gfCNCPoint5[8465] = {X 489.4800, Y 58.0000, Z -7.1667, A 0.000, B 0.000, C 0.000 }
gfCNCPoint5[8466] = {X 489.4795, Y 59.0537, Z -7.1667, A 0.000, B 0.000, C 0.000 }
gfCNCPoint5[8467] = {X 489.3596, Y 60.7976, Z -7.1667, A 0.000, B 0.000, C 0.000 }
gfCNCPoint5[8468] = {X 489.0304, Y 62.5143, Z -7.1667, A 0.000, B 0.000, C 0.000 }
gfCNCPoint5[8469] = {X 488.4968, Y 64.1788, Z -7.1667, A 0.000, B 0.000, C 0.000 }
gfCNCPoint5[8470] = {X 487.7665, Y 65.7669, Z -7.1667, A 0.000, B 0.000, C 0.000 }
gfCNCPoint5[8471] = {X 486.8501, Y 67.2554, Z -7.1667, A 0.000, B 0.000, C 0.000 }
gfCNCPoint5[8472] = {X 485.7611, Y 68.6227, Z -7.1667, A 0.000, B 0.000, C 0.000 }
gfCNCPoint5[8473] = {X 485.7614, Y 87.3811, Z -7.1667, A 0.000, B 0.000, C 0.000 }
gfCNCPoint5[8474] = {X 486.0686, Y 87.7333, Z -7.1667, A 0.000, B 0.000, C 0.000 }
gfCNCPoint5[8475] = {X 486.3643, Y 88.0951, Z -7.1667, A 0.000, B 0.000, C 0.000 }
gfCNCPoint5[8476] = {X 507.6812, Y 88.0951, Z -7.1667, A 0.000, B 0.000, C 0.000 }
gfCNCPoint5[8477] = {X 507.6812, Y 90.4951, Z -7.1667, A 0.000, B 0.000, C 0.000 }
gfCNCPoint5[8478] = {X 590.4967, Y 90.4951, Z -7.1667, A 0.000, B 0.000, C 0.000 }
gfCNCPoint5[8479] = {X 590.4967, Y 58.6615, Z -7.1667, A 0.000, B 0.000, C 0.000 }
gfCNCPoint5[8480] = {X 588.9715, Y 58.2279, Z -7.1667, A 0.000, B 0.000, C 0.000 }
gfCNCPoint5[8481] = {X 587.5052, Y 57.6246, Z -7.1667, A 0.000, B 0.000, C 0.000 }
gfCNCPoint5[8482] = {X 585.8387, Y 58.2956, Z -7.1667, A 0.000, B 0.000, C 0.000 }
gfCNCPoint5[8483] = {X 584.0999, Y 58.7477, Z -7.1667, A 0.000, B 0.000, C 0.000 }
gfCNCPoint5[8484] = {X 582.3176, Y 58.9733, Z -7.1667, A 0.000, B 0.000, C 0.000 }
gfCNCPoint5[8485] = {X 580.5210, Y 58.9689, Z -7.1667, A 0.000, B 0.000, C 0.000 }
gfCNCPoint5[8486] = {X 578.7398, Y 58.7344, Z -7.1667, A 0.000, B 0.000, C 0.000 }
gfCNCPoint5[8487] = {X 577.0034, Y 58.2738, Z -7.1667, A 0.000, B 0.000, C 0.000 }
gfCNCPoint5[8488] = {X 575.3401, Y 57.5945, Z -7.1667, A 0.000, B 0.000, C 0.000 }
gfCNCPoint5[8489] = {X 573.8813, Y 58.2035, Z -7.1667, A 0.000, B 0.000, C 0.000 }
gfCNCPoint5[8490] = {X 572.3630, Y 58.6441, Z -7.1667, A 0.000, B 0.000, C 0.000 }
gfCNCPoint5[8491] = {X 570.8048, Y 58.9107, Z -7.1667, A 0.000, B 0.000, C 0.000 }
gfCNCPoint5[8492] = {X 569.2264, Y 59.0000, Z -7.1667, A 0.000, B 0.000, C 0.000 }
gfCNCPoint5[8493] = {X 562.4443, Y 59.0000, Z -7.1667, A 0.000, B 0.000, C 0.000 }
gfCNCPoint5[8494] = {X 560.6169, Y 58.8802, Z -7.1667, A 0.000, B 0.000, C 0.000 }
gfCNCPoint5[8495] = {X 558.8208, Y 58.5230, Z -7.1667, A 0.000, B 0.000, C 0.000 }
gfCNCPoint5[8496] = {X 557.0867, Y 57.9343, Z -7.1667, A 0.000, B 0.000, C 0.000 }
gfCNCPoint5[8497] = {X 555.4443, Y 57.1244, Z -7.1667, A 0.000, B 0.000, C 0.000 }
gfCNCPoint5[8498] = {X 553.9216, Y 56.1069, Z -7.1667, A 0.000, B 0.000, C 0.000 }
gfCNCPoint5[8499] = {X 552.5448, Y 54.8995, Z -7.1667, A 0.000, B 0.000, C 0.000 }
gfCNCPoint5[8500] = {X 551.4383, Y 53.6527, Z -7.1667, A 0.000, B 0.000, C 0.000 }
gfCNCPoint5[8501] = {X 550.4879, Y 52.2832, Z -7.1667, A 0.000, B 0.000, C 0.000 }
gfCNCPoint5[8502] = {X 549.8381, Y 51.0896, Z -7.1667, A 0.000, B 0.000, C 0.000 }
gfCNCPoint5[8503] = {X 549.3070, Y 49.8386, Z -7.1667, A 0.000, B 0.000, C 0.000 }
gfCNCPoint5[8504] = {X 548.3757, Y 50.7155, Z -7.1667, A 0.000, B 0.000, C 0.000 }
gfCNCPoint5[8505] = {X 547.3054, Y 51.4159, Z -7.1667, A 0.000, B 0.000, C 0.000 }
gfCNCPoint5[8506] = {X 546.1638, Y 51.9069, Z -7.1667, A 0.000, B 0.000, C 0.000 }
gfCNCPoint5[8507] = {X 544.9553, Y 52.1968, Z -7.1667, A 0.000, B 0.000, C 0.000 }
gfCNCPoint5[8508] = {X 543.7151, Y 52.2769, Z -7.1667, A 0.000, B 0.000, C 0.000 }
gfCNCPoint5[8509] = {X 525.3425, Y 52.2772, Z -7.1667, A 0.000, B 0.000, C 0.000 }
gfCNCPoint5[8510] = {X 524.2751, Y 53.0687, Z -7.1667, A 0.000, B 0.000, C 0.000 }
gfCNCPoint5[8511] = {X 523.0839, Y 53.6575, Z -7.1667, A 0.000, B 0.000, C 0.000 }
gfCNCPoint5[8512] = {X 521.8069, Y 54.0249, Z -7.1667, A 0.000, B 0.000, C 0.000 }
gfCNCPoint5[8513] = {X 520.4849, Y 54.1591, Z -7.1667, A 0.000, B 0.000, C 0.000 }
gfCNCPoint5[8514] = {X 519.7998, Y 54.1591, Z -7.1667, A 0.000, B 0.000, C 0.000 }
gfCNCPoint5[8515] = {X 518.5529, Y 54.0515, Z -7.1667, A 0.000, B 0.000, C 0.000 }
gfCNCPoint5[8516] = {X 517.3428, Y 53.7320, Z -7.1667, A 0.000, B 0.000, C 0.000 }
gfCNCPoint5[8517] = {X 516.2054, Y 53.2099, Z -7.1667, A 0.000, B 0.000, C 0.000 }
gfCNCPoint5[8518] = {X 515.1742, Y 52.5007, Z -7.1667, A 0.000, B 0.000, C 0.000 }
gfCNCPoint5[8519] = {X 514.2797, Y 51.6254, Z -7.1667, A 0.000, B 0.000, C 0.000 }
gfCNCPoint5[8520] = {X 513.5483, Y 50.6098, Z -7.1667, A 0.000, B 0.000, C 0.000 }
gfCNCPoint5[8521] = {X 513.0017, Y 49.4839, Z -7.1667, A 0.000, B 0.000, C 0.000 }
gfCNCPoint5[8522] = {X 512.7353, Y 48.6374, Z -7.1667, A 0.000, B 0.000, C 0.000 }
gfCNCPoint5[8523] = {X 512.5739, Y 47.7649, Z -7.1667, A 0.000, B 0.000, C 0.000 }
gfCNCPoint5[8524] = {X 512.5198, Y 46.8791, Z -7.1667, A 0.000, B 0.000, C 0.000 }
gfCNCPoint5[8525] = {X 512.5198, Y 39.9011, Z -7.1667, A 0.000, B 0.000, C 0.000 }
gfCNCPoint5[8526] = {X 512.5808, Y 38.9604, Z -7.1667, A 0.000, B 0.000, C 0.000 }
gfCNCPoint5[8527] = {X 512.7629, Y 38.0355, Z -7.1667, A 0.000, B 0.000, C 0.000 }
gfCNCPoint5[8528] = {X 513.0629, Y 37.1419, Z -7.1667, A 0.000, B 0.000, C 0.000 }
gfCNCPoint5[8529] = {X 513.5586, Y 36.1533, Z -7.1667, A 0.000, B 0.000, C 0.000 }
gfCNCPoint5[8530] = {X 514.1983, Y 35.2512, Z -7.1667, A 0.000, B 0.000, C 0.000 }
gfCNCPoint5[8531] = {X 514.9672, Y 34.4564, Z -7.1667, A 0.000, B 0.000, C 0.000 }
gfCNCPoint5[8532] = {X 515.8477, Y 33.7872, Z -7.1667, A 0.000, B 0.000, C 0.000 }
gfCNCPoint5[8533] = {X 513.2419, Y 29.7561, Z -7.1667, A 0.000, B 0.000, C 0.000 }
gfCNCPoint5[8534] = {X 513.5220, Y 29.5804, Z -7.1667, A 0.000, B 0.000, C 0.000 }
gfCNCPoint5[8535] = {X 513.8068, Y 29.4125, Z -7.1667, A 0.000, B 0.000, C 0.000 }
gfCNCPoint5[8536] = {X 513.8068, Y 27.6757, Z -7.1667, A 0.000, B 0.000, C 0.000 }
gfCNCPoint5[8537] = {X 513.5219, Y 27.5014, Z -7.1667, A 0.000, B 0.000, C 0.000 }
gfCNCPoint5[8538] = {X 513.2419, Y 27.3192, Z -7.1667, A 0.000, B 0.000, C 0.000 }
gfCNCPoint5[8539] = {X 513.2419, Y 29.7561, Z -7.1667, A 0.000, B 0.000, C 0.000 }
gfCNCPoint5[8540] = {X 514.5448, Y 31.7717, Z -7.1667, A 0.000, B 0.000, C 0.000 }
gfCNCPoint5[8541] = {X 515.3550, Y 31.3019, Z -7.1667, A 0.000, B 0.000, C 0.000 }
gfCNCPoint5[8542] = {X 516.2068, Y 30.9126, Z -7.1667, A 0.000, B 0.000, C 0.000 }
gfCNCPoint5[8543] = {X 516.2068, Y 26.2046, Z -7.1667, A 0.000, B 0.000, C 0.000 }
gfCNCPoint5[8544] = {X 515.3716, Y 25.8042, Z -7.1667, A 0.000, B 0.000, C 0.000 }
gfCNCPoint5[8545] = {X 514.5784, Y 25.3258, Z -7.1667, A 0.000, B 0.000, C 0.000 }
gfCNCPoint5[8546] = {X 513.5954, Y 24.5712, Z -7.1667, A 0.000, B 0.000, C 0.000 }
gfCNCPoint5[8547] = {X 512.7167, Y 23.6971, Z -7.1667, A 0.000, B 0.000, C 0.000 }
gfCNCPoint5[8548] = {X 511.9570, Y 22.7179, Z -7.1667, A 0.000, B 0.000, C 0.000 }
gfCNCPoint5[8549] = {X 511.3286, Y 21.6497, Z -7.1667, A 0.000, B 0.000, C 0.000 }
gfCNCPoint5[8550] = {X 510.8418, Y 20.5099, Z -7.1667, A 0.000, B 0.000, C 0.000 }
gfCNCPoint5[8551] = {X 510.8420, Y 36.2322, Z -7.1667, A 0.000, B 0.000, C 0.000 }
gfCNCPoint5[8552] = {X 511.5011, Y 34.9177, Z -7.1667, A 0.000, B 0.000, C 0.000 }
gfCNCPoint5[8553] = {X 512.3517, Y 33.7182, Z -7.1667, A 0.000, B 0.000, C 0.000 }
gfCNCPoint5[8554] = {X 513.3741, Y 32.6614, Z -7.1667, A 0.000, B 0.000, C 0.000 }
gfCNCPoint5[8555] = {X 514.5448, Y 31.7717, Z -7.1667, A 0.000, B 0.000, C 0.000 }
gfCNCPoint5[8556] = {X 515.8477, Y 33.7872, Z -7.1667, A 0.000, B 0.000, C 0.000 }
gfCNCPoint5[8557] = {X 516.7441, Y 33.2935, Z -7.1667, A 0.000, B 0.000, C 0.000 }
gfCNCPoint5[8558] = {X 517.7008, Y 32.9303, Z -7.1667, A 0.000, B 0.000, C 0.000 }
gfCNCPoint5[8559] = {X 518.6990, Y 32.7048, Z -7.1667, A 0.000, B 0.000, C 0.000 }
gfCNCPoint5[8560] = {X 518.6299, Y 32.1290, Z -7.1667, A 0.000, B 0.000, C 0.000 }
gfCNCPoint5[8561] = {X 518.6068, Y 31.5494, Z -7.1667, A 0.000, B 0.000, C 0.000 }
gfCNCPoint5[8562] = {X 518.6068, Y 24.5714, Z -7.1667, A 0.000, B 0.000, C 0.000 }
gfCNCPoint5[8563] = {X 518.6080, Y 24.4373, Z -7.1667, A 0.000, B 0.000, C 0.000 }
gfCNCPoint5[8564] = {X 517.3914, Y 24.0941, Z -7.1667, A 0.000, B 0.000, C 0.000 }
gfCNCPoint5[8565] = {X 516.2525, Y 23.5455, Z -7.1667, A 0.000, B 0.000, C 0.000 }
gfCNCPoint5[8566] = {X 515.2257, Y 22.8082, Z -7.1667, A 0.000, B 0.000, C 0.000 }
gfCNCPoint5[8567] = {X 514.3419, Y 21.9045, Z -7.1667, A 0.000, B 0.000, C 0.000 }
gfCNCPoint5[8568] = {X 513.6277, Y 20.8614, Z -7.1667, A 0.000, B 0.000, C 0.000 }
gfCNCPoint5[8569] = {X 513.1048, Y 19.7105, Z -7.1667, A 0.000, B 0.000, C 0.000 }
gfCNCPoint5[8570] = {X 512.7938, Y 18.5158, Z -7.1667, A 0.000, B 0.000, C 0.000 }
gfCNCPoint5[8571] = {X 512.6891, Y 17.2857, Z -7.1667, A 0.000, B 0.000, C 0.000 }
gfCNCPoint5[8572] = {X 512.6891, Y 10.3077, Z -7.1667, A 0.000, B 0.000, C 0.000 }
gfCNCPoint5[8573] = {X 512.7002, Y 9.9057, Z -7.1667, A 0.000, B 0.000, C 0.000 }
gfCNCPoint5[8574] = {X 512.7335, Y 9.5049, Z -7.1667, A 0.000, B 0.000, C 0.000 }
gfCNCPoint5[8575] = {X 509.4593, Y 9.5049, Z -7.1667, A 0.000, B 0.000, C 0.000 }
gfCNCPoint5[8576] = {X 509.7407, Y 10.3716, Z -7.1667, A 0.000, B 0.000, C 0.000 }
gfCNCPoint5[8577] = {X 509.9113, Y 11.2668, Z -7.1667, A 0.000, B 0.000, C 0.000 }
gfCNCPoint5[8578] = {X 509.9685, Y 12.1762, Z -7.1667, A 0.000, B 0.000, C 0.000 }
gfCNCPoint5[8579] = {X 509.9682, Y 13.0462, Z -7.1667, A 0.000, B 0.000, C 0.000 }
gfCNCPoint5[8580] = {X 509.8612, Y 14.2233, Z -7.1667, A 0.000, B 0.000, C 0.000 }
gfCNCPoint5[8581] = {X 509.5651, Y 15.3676, Z -7.1667, A 0.000, B 0.000, C 0.000 }
gfCNCPoint5[8582] = {X 509.0878, Y 16.4489, Z -7.1667, A 0.000, B 0.000, C 0.000 }
gfCNCPoint5[8583] = {X 508.4418, Y 17.4387, Z -7.1667, A 0.000, B 0.000, C 0.000 }
gfCNCPoint5[8584] = {X 508.4420, Y 39.7484, Z -7.1667, A 0.000, B 0.000, C 0.000 }
gfCNCPoint5[8585] = {X 509.0898, Y 40.7415, Z -7.1667, A 0.000, B 0.000, C 0.000 }
gfCNCPoint5[8586] = {X 509.5677, Y 41.8266, Z -7.1667, A 0.000, B 0.000, C 0.000 }
gfCNCPoint5[8587] = {X 509.8632, Y 42.9748, Z -7.1667, A 0.000, B 0.000, C 0.000 }
gfCNCPoint5[8588] = {X 509.9683, Y 44.1558, Z -7.1667, A 0.000, B 0.000, C 0.000 }
gfCNCPoint5[8589] = {X 509.9685, Y 45.0000, Z -7.1667, A 0.000, B 0.000, C 0.000 }
gfCNCPoint5[8590] = {X 509.8909, Y 46.0603, Z -7.1667, A 0.000, B 0.000, C 0.000 }
gfCNCPoint5[8591] = {X 509.6596, Y 47.0980, Z -7.1667, A 0.000, B 0.000, C 0.000 }
gfCNCPoint5[8592] = {X 509.2797, Y 48.0910, Z -7.1667, A 0.000, B 0.000, C 0.000 }
gfCNCPoint5[8593] = {X 508.7593, Y 49.0180, Z -7.1667, A 0.000, B 0.000, C 0.000 }
gfCNCPoint5[8594] = {X 508.0200, Y 49.9571, Z -7.1667, A 0.000, B 0.000, C 0.000 }
gfCNCPoint5[8595] = {X 507.1371, Y 50.7626, Z -7.1667, A 0.000, B 0.000, C 0.000 }
gfCNCPoint5[8596] = {X 506.1343, Y 51.4129, Z -7.1667, A 0.000, B 0.000, C 0.000 }
gfCNCPoint5[8597] = {X 505.0386, Y 51.8902, Z -7.1667, A 0.000, B 0.000, C 0.000 }
gfCNCPoint5[8598] = {X 503.8796, Y 52.1819, Z -7.1667, A 0.000, B 0.000, C 0.000 }
gfCNCPoint5[8599] = {X 502.6885, Y 52.2800, Z -7.1667, A 0.000, B 0.000, C 0.000 }
gfCNCPoint5[8600] = {X 496.2450, Y 52.2800, Z -7.1667, A 0.000, B 0.000, C 0.000 }
gfCNCPoint5[8601] = {X 495.0845, Y 52.1869, Z -7.1667, A 0.000, B 0.000, C 0.000 }
gfCNCPoint5[8602] = {X 493.9538, Y 51.9100, Z -7.1667, A 0.000, B 0.000, C 0.000 }
gfCNCPoint5[8603] = {X 492.8816, Y 51.4564, Z -7.1667, A 0.000, B 0.000, C 0.000 }
gfCNCPoint5[8604] = {X 491.8954, Y 50.8377, Z -7.1667, A 0.000, B 0.000, C 0.000 }
gfCNCPoint5[8605] = {X 491.0204, Y 50.0697, Z -7.1667, A 0.000, B 0.000, C 0.000 }
gfCNCPoint5[8606] = {X 490.2980, Y 49.1989, Z -7.1667, A 0.000, B 0.000, C 0.000 }
gfCNCPoint5[8607] = {X 489.7192, Y 48.2267, Z -7.1667, A 0.000, B 0.000, C 0.000 }
gfCNCPoint5[8608] = {X 489.2980, Y 47.1766, Z -7.1667, A 0.000, B 0.000, C 0.000 }
gfCNCPoint5[8609] = {X 488.8769, Y 48.2267, Z -7.1667, A 0.000, B 0.000, C 0.000 }
gfCNCPoint5[8610] = {X 488.2981, Y 49.1989, Z -7.1667, A 0.000, B 0.000, C 0.000 }
gfCNCPoint5[8611] = {X 487.5756, Y 50.0697, Z -7.1667, A 0.000, B 0.000, C 0.000 }
gfCNCPoint5[8612] = {X 486.8824, Y 50.6978, Z -7.1667, A 0.000, B 0.000, C 0.000 }
gfCNCPoint5[8613] = {X 486.1145, Y 51.2318, Z -7.1667, A 0.000, B 0.000, C 0.000 }
gfCNCPoint5[8614] = {X 485.2843, Y 51.6629, Z -7.1667, A 0.000, B 0.000, C 0.000 }
gfCNCPoint5[8615] = {X 486.0586, Y 53.1385, Z -7.1667, A 0.000, B 0.000, C 0.000 }
gfCNCPoint5[8616] = {X 486.6224, Y 54.7067, Z -7.1667, A 0.000, B 0.000, C 0.000 }
gfCNCPoint5[8617] = {X 486.9651, Y 56.3375, Z -7.1667, A 0.000, B 0.000, C 0.000 }
gfCNCPoint5[8618] = {X 487.0800, Y 58.0000, Z -7.1667, A 0.000, B 0.000, C 0.000 }
gfCNCPoint5[8619] = {X 487.0796, Y 59.0339, Z -7.1667, A 0.000, B 0.000, C 0.000 }
gfCNCPoint5[8620] = {X 486.9596, Y 60.6350, Z -7.1667, A 0.000, B 0.000, C 0.000 }
gfCNCPoint5[8621] = {X 486.6284, Y 62.2061, Z -7.1667, A 0.000, B 0.000, C 0.000 }
gfCNCPoint5[8622] = {X 486.0918, Y 63.7194, Z -7.1667, A 0.000, B 0.000, C 0.000 }
gfCNCPoint5[8623] = {X 485.3591, Y 65.1481, Z -7.1667, A 0.000, B 0.000, C 0.000 }
gfCNCPoint5[8624] = {X 484.4435, Y 66.4671, Z -7.1667, A 0.000, B 0.000, C 0.000 }
gfCNCPoint5[8625] = {X 483.3611, Y 67.6530, Z -7.1667, A 0.000, B 0.000, C 0.000 }
gfCNCPoint5[8626] = {X 483.3614, Y 88.3518, Z -7.1667, A 0.000, B 0.000, C 0.000 }
gfCNCPoint5[8627] = {X 484.3105, Y 89.3721, Z -7.1667, A 0.000, B 0.000, C 0.000 }
gfCNCPoint5[8628] = {X 485.1356, Y 90.4951, Z -7.1667, A 0.000, B 0.000, C 0.000 }
gfCNCPoint5[8629] = {X 507.6812, Y 90.4951, Z -7.1667, A 0.000, B 0.000, C 0.000 }
gfCNCPoint5[8630] = {X 507.6812, Y 92.8951, Z -7.1667, A 0.000, B 0.000, C 0.000 }
gfCNCPoint5[8631] = {X 592.8967, Y 92.8951, Z -7.1667, A 0.000, B 0.000, C 0.000 }
gfCNCPoint5[8632] = {X 592.8967, Y 56.5812, Z -7.1667, A 0.000, B 0.000, C 0.000 }
gfCNCPoint5[8633] = {X 591.4811, Y 56.4128, Z -7.1667, A 0.000, B 0.000, C 0.000 }
gfCNCPoint5[8634] = {X 590.0968, Y 56.0721, Z -7.1667, A 0.000, B 0.000, C 0.000 }
gfCNCPoint5[8635] = {X 588.7648, Y 55.5641, Z -7.1667, A 0.000, B 0.000, C 0.000 }
gfCNCPoint5[8636] = {X 587.5052, Y 54.8965, Z -7.1667, A 0.000, B 0.000, C 0.000 }
gfCNCPoint5[8637] = {X 586.9690, Y 55.2051, Z -7.1667, A 0.000, B 0.000, C 0.000 }
gfCNCPoint5[8638] = {X 586.4171, Y 55.4846, Z -7.1667, A 0.000, B 0.000, C 0.000 }
gfCNCPoint5[8639] = {X 584.8782, Y 56.0830, Z -7.1667, A 0.000, B 0.000, C 0.000 }
gfCNCPoint5[8640] = {X 583.2699, Y 56.4570, Z -7.1667, A 0.000, B 0.000, C 0.000 }
gfCNCPoint5[8641] = {X 581.6248, Y 56.5987, Z -7.1667, A 0.000, B 0.000, C 0.000 }
gfCNCPoint5[8642] = {X 579.9763, Y 56.5055, Z -7.1667, A 0.000, B 0.000, C 0.000 }
gfCNCPoint5[8643] = {X 578.3577, Y 56.1792, Z -7.1667, A 0.000, B 0.000, C 0.000 }
gfCNCPoint5[8644] = {X 576.8018, Y 55.6263, Z -7.1667, A 0.000, B 0.000, C 0.000 }
gfCNCPoint5[8645] = {X 575.3401, Y 54.8581, Z -7.1667, A 0.000, B 0.000, C 0.000 }
gfCNCPoint5[8646] = {X 573.9176, Y 55.6091, Z -7.1667, A 0.000, B 0.000, C 0.000 }
gfCNCPoint5[8647] = {X 572.4049, Y 56.1560, Z -7.1667, A 0.000, B 0.000, C 0.000 }
gfCNCPoint5[8648] = {X 570.8311, Y 56.4885, Z -7.1667, A 0.000, B 0.000, C 0.000 }
gfCNCPoint5[8649] = {X 569.2264, Y 56.6000, Z -7.1667, A 0.000, B 0.000, C 0.000 }
gfCNCPoint5[8650] = {X 562.4443, Y 56.6000, Z -7.1667, A 0.000, B 0.000, C 0.000 }
gfCNCPoint5[8651] = {X 560.9302, Y 56.5008, Z -7.1667, A 0.000, B 0.000, C 0.000 }
gfCNCPoint5[8652] = {X 559.4420, Y 56.2047, Z -7.1667, A 0.000, B 0.000, C 0.000 }
gfCNCPoint5[8653] = {X 558.0052, Y 55.7170, Z -7.1667, A 0.000, B 0.000, C 0.000 }
gfCNCPoint5[8654] = {X 556.6443, Y 55.0459, Z -7.1667, A 0.000, B 0.000, C 0.000 }
gfCNCPoint5[8655] = {X 555.3827, Y 54.2029, Z -7.1667, A 0.000, B 0.000, C 0.000 }
gfCNCPoint5[8656] = {X 554.2419, Y 53.2024, Z -7.1667, A 0.000, B 0.000, C 0.000 }
gfCNCPoint5[8657] = {X 553.4046, Y 52.2694, Z -7.1667, A 0.000, B 0.000, C 0.000 }
gfCNCPoint5[8658] = {X 552.6729, Y 51.2514, Z -7.1667, A 0.000, B 0.000, C 0.000 }
gfCNCPoint5[8659] = {X 552.0553, Y 50.1604, Z -7.1667, A 0.000, B 0.000, C 0.000 }
gfCNCPoint5[8660] = {X 551.5591, Y 49.0091, Z -7.1667, A 0.000, B 0.000, C 0.000 }
gfCNCPoint5[8661] = {X 551.1638, Y 47.7039, Z -7.1667, A 0.000, B 0.000, C 0.000 }
gfCNCPoint5[8662] = {X 550.9245, Y 46.3614, Z -7.1667, A 0.000, B 0.000, C 0.000 }
gfCNCPoint5[8663] = {X 550.8443, Y 45.0000, Z -7.1667, A 0.000, B 0.000, C 0.000 }
gfCNCPoint5[8664] = {X 550.8443, Y 44.0403, Z -7.1667, A 0.000, B 0.000, C 0.000 }
gfCNCPoint5[8665] = {X 550.9580, Y 42.4569, Z -7.1667, A 0.000, B 0.000, C 0.000 }
gfCNCPoint5[8666] = {X 551.2863, Y 40.9037, Z -7.1667, A 0.000, B 0.000, C 0.000 }
gfCNCPoint5[8667] = {X 551.8231, Y 39.4097, Z -7.1667, A 0.000, B 0.000, C 0.000 }
gfCNCPoint5[8668] = {X 549.6250, Y 38.4460, Z -7.1667, A 0.000, B 0.000, C 0.000 }
gfCNCPoint5[8669] = {X 549.7927, Y 38.0781, Z -7.1667, A 0.000, B 0.000, C 0.000 }
gfCNCPoint5[8670] = {X 549.9709, Y 37.7152, Z -7.1667, A 0.000, B 0.000, C 0.000 }
gfCNCPoint5[8671] = {X 549.9710, Y 16.9522, Z -7.1667, A 0.000, B 0.000, C 0.000 }
gfCNCPoint5[8672] = {X 549.8033, Y 17.1983, Z -7.1667, A 0.000, B 0.000, C 0.000 }
gfCNCPoint5[8673] = {X 549.6257, Y 17.4374, Z -7.1667, A 0.000, B 0.000, C 0.000 }
gfCNCPoint5[8674] = {X 549.6250, Y 38.4460, Z -7.1667, A 0.000, B 0.000, C 0.000 }
gfCNCPoint5[8675] = {X 551.8231, Y 39.4097, Z -7.1667, A 0.000, B 0.000, C 0.000 }
gfCNCPoint5[8676] = {X 552.0827, Y 38.8574, Z -7.1667, A 0.000, B 0.000, C 0.000 }
gfCNCPoint5[8677] = {X 552.3709, Y 38.3195, Z -7.1667, A 0.000, B 0.000, C 0.000 }
gfCNCPoint5[8678] = {X 552.3710, Y 11.6864, Z -7.1667, A 0.000, B 0.000, C 0.000 }
gfCNCPoint5[8679] = {X 551.6701, Y 10.2325, Z -7.1667, A 0.000, B 0.000, C 0.000 }
gfCNCPoint5[8680] = {X 551.1778, Y 8.6954, Z -7.1667, A 0.000, B 0.000, C 0.000 }
gfCNCPoint5[8681] = {X 550.9035, Y 7.1049, Z -7.1667, A 0.000, B 0.000, C 0.000 }
gfCNCPoint5[8682] = {X 524.2927, Y 7.1049, Z -7.1667, A 0.000, B 0.000, C 0.000 }
gfCNCPoint5[8683] = {X 524.3782, Y 7.2059, Z -7.1667, A 0.000, B 0.000, C 0.000 }
gfCNCPoint5[8684] = {X 524.4609, Y 7.3092, Z -7.1667, A 0.000, B 0.000, C 0.000 }
gfCNCPoint5[8685] = {X 543.7426, Y 7.3096, Z -7.1667, A 0.000, B 0.000, C 0.000 }
gfCNCPoint5[8686] = {X 544.7121, Y 7.3817, Z -7.1667, A 0.000, B 0.000, C 0.000 }
gfCNCPoint5[8687] = {X 545.6480, Y 7.6444, Z -7.1667, A 0.000, B 0.000, C 0.000 }
gfCNCPoint5[8688] = {X 546.5134, Y 8.0872, Z -7.1667, A 0.000, B 0.000, C 0.000 }
gfCNCPoint5[8689] = {X 547.2740, Y 8.6926, Z -7.1667, A 0.000, B 0.000, C 0.000 }
gfCNCPoint5[8690] = {X 547.8996, Y 9.4366, Z -7.1667, A 0.000, B 0.000, C 0.000 }
gfCNCPoint5[8691] = {X 548.3656, Y 10.2898, Z -7.1667, A 0.000, B 0.000, C 0.000 }
gfCNCPoint5[8692] = {X 548.6533, Y 11.2184, Z -7.1667, A 0.000, B 0.000, C 0.000 }
gfCNCPoint5[8693] = {X 548.7514, Y 12.1856, Z -7.1667, A 0.000, B 0.000, C 0.000 }
gfCNCPoint5[8694] = {X 548.7512, Y 13.0237, Z -7.1667, A 0.000, B 0.000, C 0.000 }
gfCNCPoint5[8695] = {X 548.6554, Y 13.9414, Z -7.1667, A 0.000, B 0.000, C 0.000 }
gfCNCPoint5[8696] = {X 548.3885, Y 14.8247, Z -7.1667, A 0.000, B 0.000, C 0.000 }
gfCNCPoint5[8697] = {X 547.9601, Y 15.6420, Z -7.1667, A 0.000, B 0.000, C 0.000 }
gfCNCPoint5[8698] = {X 547.6189, Y 16.1039, Z -7.1667, A 0.000, B 0.000, C 0.000 }
gfCNCPoint5[8699] = {X 547.2258, Y 16.5224, Z -7.1667, A 0.000, B 0.000, C 0.000 }
gfCNCPoint5[8700] = {X 547.2250, Y 40.6636, Z -7.1667, A 0.000, B 0.000, C 0.000 }
gfCNCPoint5[8701] = {X 547.8659, Y 41.4055, Z -7.1667, A 0.000, B 0.000, C 0.000 }
gfCNCPoint5[8702] = {X 548.3456, Y 42.2605, Z -7.1667, A 0.000, B 0.000, C 0.000 }
gfCNCPoint5[8703] = {X 548.6448, Y 43.1941, Z -7.1667, A 0.000, B 0.000, C 0.000 }
gfCNCPoint5[8704] = {X 548.7513, Y 44.1687, Z -7.1667, A 0.000, B 0.000, C 0.000 }
gfCNCPoint5[8705] = {X 548.7514, Y 45.0006, Z -7.1667, A 0.000, B 0.000, C 0.000 }
gfCNCPoint5[8706] = {X 548.6700, Y 45.8824, Z -7.1667, A 0.000, B 0.000, C 0.000 }
gfCNCPoint5[8707] = {X 548.4306, Y 46.7350, Z -7.1667, A 0.000, B 0.000, C 0.000 }
gfCNCPoint5[8708] = {X 548.0413, Y 47.5304, Z -7.1667, A 0.000, B 0.000, C 0.000 }
gfCNCPoint5[8709] = {X 547.5147, Y 48.2424, Z -7.1667, A 0.000, B 0.000, C 0.000 }
gfCNCPoint5[8710] = {X 546.7291, Y 48.9521, Z -7.1667, A 0.000, B 0.000, C 0.000 }
gfCNCPoint5[8711] = {X 545.8090, Y 49.4759, Z -7.1667, A 0.000, B 0.000, C 0.000 }
gfCNCPoint5[8712] = {X 544.7976, Y 49.7890, Z -7.1667, A 0.000, B 0.000, C 0.000 }
gfCNCPoint5[8713] = {X 543.7426, Y 49.8769, Z -7.1667, A 0.000, B 0.000, C 0.000 }
gfCNCPoint5[8714] = {X 524.3239, Y 49.8773, Z -7.1667, A 0.000, B 0.000, C 0.000 }
gfCNCPoint5[8715] = {X 523.7110, Y 50.5161, Z -7.1667, A 0.000, B 0.000, C 0.000 }
gfCNCPoint5[8716] = {X 522.9957, Y 51.0377, Z -7.1667, A 0.000, B 0.000, C 0.000 }
gfCNCPoint5[8717] = {X 522.2001, Y 51.4260, Z -7.1667, A 0.000, B 0.000, C 0.000 }
gfCNCPoint5[8718] = {X 521.3488, Y 51.6690, Z -7.1667, A 0.000, B 0.000, C 0.000 }
gfCNCPoint5[8719] = {X 520.4681, Y 51.7591, Z -7.1667, A 0.000, B 0.000, C 0.000 }
gfCNCPoint5[8720] = {X 519.7998, Y 51.7591, Z -7.1667, A 0.000, B 0.000, C 0.000 }
gfCNCPoint5[8721] = {X 518.8477, Y 51.6654, Z -7.1667, A 0.000, B 0.000, C 0.000 }
gfCNCPoint5[8722] = {X 517.9323, Y 51.3877, Z -7.1667, A 0.000, B 0.000, C 0.000 }
gfCNCPoint5[8723] = {X 517.0886, Y 50.9367, Z -7.1667, A 0.000, B 0.000, C 0.000 }
gfCNCPoint5[8724] = {X 516.3491, Y 50.3298, Z -7.1667, A 0.000, B 0.000, C 0.000 }
gfCNCPoint5[8725] = {X 515.7422, Y 49.5903, Z -7.1667, A 0.000, B 0.000, C 0.000 }
gfCNCPoint5[8726] = {X 515.2912, Y 48.7466, Z -7.1667, A 0.000, B 0.000, C 0.000 }
gfCNCPoint5[8727] = {X 515.0135, Y 47.8312, Z -7.1667, A 0.000, B 0.000, C 0.000 }
gfCNCPoint5[8728] = {X 514.9198, Y 46.8791, Z -7.1667, A 0.000, B 0.000, C 0.000 }
gfCNCPoint5[8729] = {X 514.9198, Y 39.9011, Z -7.1667, A 0.000, B 0.000, C 0.000 }
gfCNCPoint5[8730] = {X 515.0197, Y 38.9186, Z -7.1667, A 0.000, B 0.000, C 0.000 }
gfCNCPoint5[8731] = {X 515.3154, Y 37.9764, Z -7.1667, A 0.000, B 0.000, C 0.000 }
gfCNCPoint5[8732] = {X 515.7947, Y 37.1129, Z -7.1667, A 0.000, B 0.000, C 0.000 }
gfCNCPoint5[8733] = {X 516.4381, Y 36.3637, Z -7.1667, A 0.000, B 0.000, C 0.000 }
gfCNCPoint5[8734] = {X 517.2191, Y 35.7593, Z -7.1667, A 0.000, B 0.000, C 0.000 }
gfCNCPoint5[8735] = {X 518.1058, Y 35.3245, Z -7.1667, A 0.000, B 0.000, C 0.000 }
gfCNCPoint5[8736] = {X 519.0619, Y 35.0772, Z -7.1667, A 0.000, B 0.000, C 0.000 }
gfCNCPoint5[8737] = {X 519.4084, Y 35.0368, Z -7.1667, A 0.000, B 0.000, C 0.000 }
gfCNCPoint5[8738] = {X 519.7568, Y 35.0213, Z -7.1667, A 0.000, B 0.000, C 0.000 }
gfCNCPoint5[8739] = {X 520.5345, Y 35.0216, Z -7.1667, A 0.000, B 0.000, C 0.000 }
gfCNCPoint5[8740] = {X 521.4082, Y 35.1125, Z -7.1667, A 0.000, B 0.000, C 0.000 }
gfCNCPoint5[8741] = {X 522.2515, Y 35.3586, Z -7.1667, A 0.000, B 0.000, C 0.000 }
gfCNCPoint5[8742] = {X 523.0370, Y 35.7519, Z -7.1667, A 0.000, B 0.000, C 0.000 }
gfCNCPoint5[8743] = {X 523.7392, Y 36.2797, Z -7.1667, A 0.000, B 0.000, C 0.000 }
gfCNCPoint5[8744] = {X 524.3355, Y 36.9248, Z -7.1667, A 0.000, B 0.000, C 0.000 }
gfCNCPoint5[8745] = {X 534.0719, Y 36.9251, Z -7.1667, A 0.000, B 0.000, C 0.000 }
gfCNCPoint5[8746] = {X 534.0719, Y 34.5262, Z -7.1667, A 0.000, B 0.000, C 0.000 }
gfCNCPoint5[8747] = {X 530.3955, Y 34.5260, Z -7.1667, A 0.000, B 0.000, C 0.000 }
gfCNCPoint5[8748] = {X 529.7957, Y 35.1743, Z -7.1667, A 0.000, B 0.000, C 0.000 }
gfCNCPoint5[8749] = {X 529.0887, Y 35.7039, Z -7.1667, A 0.000, B 0.000, C 0.000 }
gfCNCPoint5[8750] = {X 528.2979, Y 36.0973, Z -7.1667, A 0.000, B 0.000, C 0.000 }
gfCNCPoint5[8751] = {X 527.4492, Y 36.3418, Z -7.1667, A 0.000, B 0.000, C 0.000 }
gfCNCPoint5[8752] = {X 526.5703, Y 36.4293, Z -7.1667, A 0.000, B 0.000, C 0.000 }
gfCNCPoint5[8753] = {X 525.8868, Y 36.4294, Z -7.1667, A 0.000, B 0.000, C 0.000 }
gfCNCPoint5[8754] = {X 524.9094, Y 36.3306, Z -7.1667, A 0.000, B 0.000, C 0.000 }
gfCNCPoint5[8755] = {X 523.9717, Y 36.0380, Z -7.1667, A 0.000, B 0.000, C 0.000 }
gfCNCPoint5[8756] = {X 523.1116, Y 35.5636, Z -7.1667, A 0.000, B 0.000, C 0.000 }
gfCNCPoint5[8757] = {X 522.3639, Y 34.9265, Z -7.1667, A 0.000, B 0.000, C 0.000 }
gfCNCPoint5[8758] = {X 521.7590, Y 34.1525, Z -7.1667, A 0.000, B 0.000, C 0.000 }
gfCNCPoint5[8759] = {X 521.3213, Y 33.2731, Z -7.1667, A 0.000, B 0.000, C 0.000 }
gfCNCPoint5[8760] = {X 521.0686, Y 32.3239, Z -7.1667, A 0.000, B 0.000, C 0.000 }
gfCNCPoint5[8761] = {X 521.0222, Y 31.9379, Z -7.1667, A 0.000, B 0.000, C 0.000 }
gfCNCPoint5[8762] = {X 521.0068, Y 31.5494, Z -7.1667, A 0.000, B 0.000, C 0.000 }
gfCNCPoint5[8763] = {X 521.0076, Y 24.4815, Z -7.1667, A 0.000, B 0.000, C 0.000 }
gfCNCPoint5[8764] = {X 521.0984, Y 23.6300, Z -7.1667, A 0.000, B 0.000, C 0.000 }
gfCNCPoint5[8765] = {X 521.3368, Y 22.8074, Z -7.1667, A 0.000, B 0.000, C 0.000 }
gfCNCPoint5[8766] = {X 521.7152, Y 22.0391, Z -7.1667, A 0.000, B 0.000, C 0.000 }
gfCNCPoint5[8767] = {X 521.1864, Y 22.1316, Z -7.1667, A 0.000, B 0.000, C 0.000 }
gfCNCPoint5[8768] = {X 520.6505, Y 22.1656, Z -7.1667, A 0.000, B 0.000, C 0.000 }
gfCNCPoint5[8769] = {X 519.9691, Y 22.1657, Z -7.1667, A 0.000, B 0.000, C 0.000 }
gfCNCPoint5[8770] = {X 519.5109, Y 22.1442, Z -7.1667, A 0.000, B 0.000, C 0.000 }
gfCNCPoint5[8771] = {X 519.0567, Y 22.0797, Z -7.1667, A 0.000, B 0.000, C 0.000 }
gfCNCPoint5[8772] = {X 518.1336, Y 21.8074, Z -7.1667, A 0.000, B 0.000, C 0.000 }
gfCNCPoint5[8773] = {X 517.2820, Y 21.3592, Z -7.1667, A 0.000, B 0.000, C 0.000 }
gfCNCPoint5[8774] = {X 516.5348, Y 20.7527, Z -7.1667, A 0.000, B 0.000, C 0.000 }
gfCNCPoint5[8775] = {X 515.9212, Y 20.0113, Z -7.1667, A 0.000, B 0.000, C 0.000 }
gfCNCPoint5[8776] = {X 515.4650, Y 19.1639, Z -7.1667, A 0.000, B 0.000, C 0.000 }
gfCNCPoint5[8777] = {X 515.1840, Y 18.2434, Z -7.1667, A 0.000, B 0.000, C 0.000 }
gfCNCPoint5[8778] = {X 515.0891, Y 17.2857, Z -7.1667, A 0.000, B 0.000, C 0.000 }
gfCNCPoint5[8779] = {X 515.0891, Y 10.3077, Z -7.1667, A 0.000, B 0.000, C 0.000 }
gfCNCPoint5[8780] = {X 515.0966, Y 10.0382, Z -7.1667, A 0.000, B 0.000, C 0.000 }
gfCNCPoint5[8781] = {X 515.1189, Y 9.7695, Z -7.1667, A 0.000, B 0.000, C 0.000 }
gfCNCPoint5[8782] = {X 515.3252, Y 8.8083, Z -7.1667, A 0.000, B 0.000, C 0.000 }
gfCNCPoint5[8783] = {X 515.7200, Y 7.9079, Z -7.1667, A 0.000, B 0.000, C 0.000 }
gfCNCPoint5[8784] = {X 516.2872, Y 7.1049, Z -7.1667, A 0.000, B 0.000, C 0.000 }
gfCNCPoint5[8785] = {X 516.6494, Y 7.4199, Z -7.1667, A 0.000, B 0.000, C 0.000 }
gfCNCPoint5[8786] = {X 517.3374, Y 6.7815, Z -7.1667, A 0.000, B 0.000, C 0.000 }
gfCNCPoint5[8787] = {X 518.1452, Y 6.3035, Z -7.1667, A 0.000, B 0.000, C 0.000 }
gfCNCPoint5[8788] = {X 519.0360, Y 6.0078, Z -7.1667, A 0.000, B 0.000, C 0.000 }
gfCNCPoint5[8789] = {X 519.9692, Y 5.9077, Z -7.1667, A 0.000, B 0.000, C 0.000 }
gfCNCPoint5[8790] = {X 520.6509, Y 5.9079, Z -7.1667, A 0.000, B 0.000, C 0.000 }
gfCNCPoint5[8791] = {X 521.4831, Y 5.9950, Z -7.1667, A 0.000, B 0.000, C 0.000 }
gfCNCPoint5[8792] = {X 522.2837, Y 6.2381, Z -7.1667, A 0.000, B 0.000, C 0.000 }
gfCNCPoint5[8793] = {X 523.0239, Y 6.6284, Z -7.1667, A 0.000, B 0.000, C 0.000 }
gfCNCPoint5[8794] = {X 523.6767, Y 7.1518, Z -7.1667, A 0.000, B 0.000, C 0.000 }
gfCNCPoint5[8795] = {X 524.2187, Y 7.7892, Z -7.1667, A 0.000, B 0.000, C 0.000 }
gfCNCPoint5[8796] = {X 543.7489, Y 7.7896, Z -7.1667, A 0.000, B 0.000, C 0.000 }
gfCNCPoint5[8797] = {X 544.7472, Y 7.8769, Z -7.1667, A 0.000, B 0.000, C 0.000 }
gfCNCPoint5[8798] = {X 545.7000, Y 8.1876, Z -7.1667, A 0.000, B 0.000, C 0.000 }
gfCNCPoint5[8799] = {X 546.5579, Y 8.7057, Z -7.1667, A 0.000, B 0.000, C 0.000 }
gfCNCPoint5[8800] = {X 547.2764, Y 9.4042, Z -7.1667, A 0.000, B 0.000, C 0.000 }
gfCNCPoint5[8801] = {X 547.8185, Y 10.2471, Z -7.1667, A 0.000, B 0.000, C 0.000 }
gfCNCPoint5[8802] = {X 548.1560, Y 11.1908, Z -7.1667, A 0.000, B 0.000, C 0.000 }
gfCNCPoint5[8803] = {X 548.2714, Y 12.1863, Z -7.1667, A 0.000, B 0.000, C 0.000 }
gfCNCPoint5[8804] = {X 548.2712, Y 13.0233, Z -7.1667, A 0.000, B 0.000, C 0.000 }
gfCNCPoint5[8805] = {X 548.1630, Y 13.9487, Z -7.1667, A 0.000, B 0.000, C 0.000 }
gfCNCPoint5[8806] = {X 547.8624, Y 14.8306, Z -7.1667, A 0.000, B 0.000, C 0.000 }
gfCNCPoint5[8807] = {X 547.3828, Y 15.6295, Z -7.1667, A 0.000, B 0.000, C 0.000 }
gfCNCPoint5[8808] = {X 546.7458, Y 16.3094, Z -7.1667, A 0.000, B 0.000, C 0.000 }
gfCNCPoint5[8809] = {X 546.7450, Y 40.8767, Z -7.1667, A 0.000, B 0.000, C 0.000 }
gfCNCPoint5[8810] = {X 547.3891, Y 41.5658, Z -7.1667, A 0.000, B 0.000, C 0.000 }
gfCNCPoint5[8811] = {X 547.8717, Y 42.3763, Z -7.1667, A 0.000, B 0.000, C 0.000 }
gfCNCPoint5[8812] = {X 548.1703, Y 43.2710, Z -7.1667, A 0.000, B 0.000, C 0.000 }
gfCNCPoint5[8813] = {X 548.2714, Y 44.2089, Z -7.1667, A 0.000, B 0.000, C 0.000 }
gfCNCPoint5[8814] = {X 548.2714, Y 45.0006, Z -7.1667, A 0.000, B 0.000, C 0.000 }
gfCNCPoint5[8815] = {X 548.1559, Y 45.9960, Z -7.1667, A 0.000, B 0.000, C 0.000 }
gfCNCPoint5[8816] = {X 547.8184, Y 46.9396, Z -7.1667, A 0.000, B 0.000, C 0.000 }
gfCNCPoint5[8817] = {X 547.2764, Y 47.7825, Z -7.1667, A 0.000, B 0.000, C 0.000 }
gfCNCPoint5[8818] = {X 546.5578, Y 48.4810, Z -7.1667, A 0.000, B 0.000, C 0.000 }
gfCNCPoint5[8819] = {X 545.6999, Y 48.9990, Z -7.1667, A 0.000, B 0.000, C 0.000 }
gfCNCPoint5[8820] = {X 544.7472, Y 49.3097, Z -7.1667, A 0.000, B 0.000, C 0.000 }
gfCNCPoint5[8821] = {X 543.7489, Y 49.3969, Z -7.1667, A 0.000, B 0.000, C 0.000 }
gfCNCPoint5[8822] = {X 524.0866, Y 49.3973, Z -7.1667, A 0.000, B 0.000, C 0.000 }
gfCNCPoint5[8823] = {X 523.5298, Y 50.0322, Z -7.1667, A 0.000, B 0.000, C 0.000 }
gfCNCPoint5[8824] = {X 522.8653, Y 50.5535, Z -7.1667, A 0.000, B 0.000, C 0.000 }
gfCNCPoint5[8825] = {X 522.1160, Y 50.9432, Z -7.1667, A 0.000, B 0.000, C 0.000 }
gfCNCPoint5[8826] = {X 521.3077, Y 51.1878, Z -7.1667, A 0.000, B 0.000, C 0.000 }
gfCNCPoint5[8827] = {X 520.4681, Y 51.2791, Z -7.1667, A 0.000, B 0.000, C 0.000 }
gfCNCPoint5[8828] = {X 519.7998, Y 51.2791, Z -7.1667, A 0.000, B 0.000, C 0.000 }
gfCNCPoint5[8829] = {X 518.8207, Y 51.1688, Z -7.1667, A 0.000, B 0.000, C 0.000 }
gfCNCPoint5[8830] = {X 517.8907, Y 50.8434, Z -7.1667, A 0.000, B 0.000, C 0.000 }
gfCNCPoint5[8831] = {X 517.0564, Y 50.3192, Z -7.1667, A 0.000, B 0.000, C 0.000 }
gfCNCPoint5[8832] = {X 516.3597, Y 49.6225, Z -7.1667, A 0.000, B 0.000, C 0.000 }
gfCNCPoint5[8833] = {X 515.8355, Y 48.7882, Z -7.1667, A 0.000, B 0.000, C 0.000 }
gfCNCPoint5[8834] = {X 515.5101, Y 47.8582, Z -7.1667, A 0.000, B 0.000, C 0.000 }
gfCNCPoint5[8835] = {X 515.3998, Y 46.8791, Z -7.1667, A 0.000, B 0.000, C 0.000 }
gfCNCPoint5[8836] = {X 515.3998, Y 39.9011, Z -7.1667, A 0.000, B 0.000, C 0.000 }
gfCNCPoint5[8837] = {X 515.5101, Y 38.9220, Z -7.1667, A 0.000, B 0.000, C 0.000 }
gfCNCPoint5[8838] = {X 515.8355, Y 37.9920, Z -7.1667, A 0.000, B 0.000, C 0.000 }
gfCNCPoint5[8839] = {X 516.3597, Y 37.1577, Z -7.1667, A 0.000, B 0.000, C 0.000 }
gfCNCPoint5[8840] = {X 517.0564, Y 36.4610, Z -7.1667, A 0.000, B 0.000, C 0.000 }
gfCNCPoint5[8841] = {X 517.8907, Y 35.9368, Z -7.1667, A 0.000, B 0.000, C 0.000 }
gfCNCPoint5[8842] = {X 518.8207, Y 35.6114, Z -7.1667, A 0.000, B 0.000, C 0.000 }
gfCNCPoint5[8843] = {X 519.7998, Y 35.5011, Z -7.1667, A 0.000, B 0.000, C 0.000 }
gfCNCPoint5[8844] = {X 520.5280, Y 35.5015, Z -7.1667, A 0.000, B 0.000, C 0.000 }
gfCNCPoint5[8845] = {X 521.3612, Y 35.5927, Z -7.1667, A 0.000, B 0.000, C 0.000 }
gfCNCPoint5[8846] = {X 522.1620, Y 35.8402, Z -7.1667, A 0.000, B 0.000, C 0.000 }
gfCNCPoint5[8847] = {X 522.9013, Y 36.2351, Z -7.1667, A 0.000, B 0.000, C 0.000 }
gfCNCPoint5[8848] = {X 523.5524, Y 36.7630, Z -7.1667, A 0.000, B 0.000, C 0.000 }
gfCNCPoint5[8849] = {X 524.0915, Y 37.4048, Z -7.1667, A 0.000, B 0.000, C 0.000 }
gfCNCPoint5[8850] = {X 534.5519, Y 37.4051, Z -7.1667, A 0.000, B 0.000, C 0.000 }
gfCNCPoint5[8851] = {X 534.5519, Y 34.0462, Z -7.1667, A 0.000, B 0.000, C 0.000 }
gfCNCPoint5[8852] = {X 530.1516, Y 34.0460, Z -7.1667, A 0.000, B 0.000, C 0.000 }
gfCNCPoint5[8853] = {X 529.6039, Y 34.6961, Z -7.1667, A 0.000, B 0.000, C 0.000 }
gfCNCPoint5[8854] = {X 528.9414, Y 35.2288, Z -7.1667, A 0.000, B 0.000, C 0.000 }
gfCNCPoint5[8855] = {X 528.1889, Y 35.6241, Z -7.1667, A 0.000, B 0.000, C 0.000 }
gfCNCPoint5[8856] = {X 527.3744, Y 35.8674, Z -7.1667, A 0.000, B 0.000, C 0.000 }
gfCNCPoint5[8857] = {X 526.5283, Y 35.9495, Z -7.1667, A 0.000, B 0.000, C 0.000 }
gfCNCPoint5[8858] = {X 525.8868, Y 35.9495, Z -7.1667, A 0.000, B 0.000, C 0.000 }
gfCNCPoint5[8859] = {X 524.9077, Y 35.8391, Z -7.1667, A 0.000, B 0.000, C 0.000 }
gfCNCPoint5[8860] = {X 523.9777, Y 35.5137, Z -7.1667, A 0.000, B 0.000, C 0.000 }
gfCNCPoint5[8861] = {X 523.1434, Y 34.9895, Z -7.1667, A 0.000, B 0.000, C 0.000 }
gfCNCPoint5[8862] = {X 522.4467, Y 34.2928, Z -7.1667, A 0.000, B 0.000, C 0.000 }
gfCNCPoint5[8863] = {X 521.9225, Y 33.4585, Z -7.1667, A 0.000, B 0.000, C 0.000 }
gfCNCPoint5[8864] = {X 521.5971, Y 32.5285, Z -7.1667, A 0.000, B 0.000, C 0.000 }
gfCNCPoint5[8865] = {X 521.4868, Y 31.5495, Z -7.1667, A 0.000, B 0.000, C 0.000 }
gfCNCPoint5[8866] = {X 521.4868, Y 24.5714, Z -7.1667, A 0.000, B 0.000, C 0.000 }
gfCNCPoint5[8867] = {X 521.5971, Y 23.5923, Z -7.1667, A 0.000, B 0.000, C 0.000 }
gfCNCPoint5[8868] = {X 521.9225, Y 22.6623, Z -7.1667, A 0.000, B 0.000, C 0.000 }
gfCNCPoint5[8869] = {X 522.4467, Y 21.8281, Z -7.1667, A 0.000, B 0.000, C 0.000 }
gfCNCPoint5[8870] = {X 523.1434, Y 21.1314, Z -7.1667, A 0.000, B 0.000, C 0.000 }
gfCNCPoint5[8871] = {X 523.9777, Y 20.6072, Z -7.1667, A 0.000, B 0.000, C 0.000 }
gfCNCPoint5[8872] = {X 524.9077, Y 20.2817, Z -7.1667, A 0.000, B 0.000, C 0.000 }
gfCNCPoint5[8873] = {X 525.8868, Y 20.1714, Z -7.1667, A 0.000, B 0.000, C 0.000 }
gfCNCPoint5[8874] = {X 526.5702, Y 20.1716, Z -7.1667, A 0.000, B 0.000, C 0.000 }
gfCNCPoint5[8875] = {X 527.2694, Y 20.2343, Z -7.1667, A 0.000, B 0.000, C 0.000 }
gfCNCPoint5[8876] = {X 527.9497, Y 20.4073, Z -7.1667, A 0.000, B 0.000, C 0.000 }
gfCNCPoint5[8877] = {X 528.5939, Y 20.6864, Z -7.1667, A 0.000, B 0.000, C 0.000 }
gfCNCPoint5[8878] = {X 528.8192, Y 20.2625, Z -7.1667, A 0.000, B 0.000, C 0.000 }
gfCNCPoint5[8879] = {X 534.0719, Y 20.2626, Z -7.1667, A 0.000, B 0.000, C 0.000 }
gfCNCPoint5[8880] = {X 534.0719, Y 21.5730, Z -7.1667, A 0.000, B 0.000, C 0.000 }
gfCNCPoint5[8881] = {X 530.3786, Y 21.5729, Z -7.1667, A 0.000, B 0.000, C 0.000 }
gfCNCPoint5[8882] = {X 529.6680, Y 20.8355, Z -7.1667, A 0.000, B 0.000, C 0.000 }
gfCNCPoint5[8883] = {X 528.8192, Y 20.2625, Z -7.1667, A 0.000, B 0.000, C 0.000 }
gfCNCPoint5[8884] = {X 528.5939, Y 20.6864, Z -7.1667, A 0.000, B 0.000, C 0.000 }
gfCNCPoint5[8885] = {X 529.1780, Y 21.0586, Z -7.1667, A 0.000, B 0.000, C 0.000 }
gfCNCPoint5[8886] = {X 529.6964, Y 21.5179, Z -7.1667, A 0.000, B 0.000, C 0.000 }
gfCNCPoint5[8887] = {X 530.1364, Y 22.0529, Z -7.1667, A 0.000, B 0.000, C 0.000 }
gfCNCPoint5[8888] = {X 534.5519, Y 22.0531, Z -7.1667, A 0.000, B 0.000, C 0.000 }
gfCNCPoint5[8889] = {X 534.5519, Y 19.7826, Z -7.1667, A 0.000, B 0.000, C 0.000 }
gfCNCPoint5[8890] = {X 524.2338, Y 19.7825, Z -7.1667, A 0.000, B 0.000, C 0.000 }
gfCNCPoint5[8891] = {X 523.6861, Y 20.4325, Z -7.1667, A 0.000, B 0.000, C 0.000 }
gfCNCPoint5[8892] = {X 523.0237, Y 20.9651, Z -7.1667, A 0.000, B 0.000, C 0.000 }
gfCNCPoint5[8893] = {X 522.2712, Y 21.3604, Z -7.1667, A 0.000, B 0.000, C 0.000 }
gfCNCPoint5[8894] = {X 521.4568, Y 21.6036, Z -7.1667, A 0.000, B 0.000, C 0.000 }
gfCNCPoint5[8895] = {X 520.6107, Y 21.6857, Z -7.1667, A 0.000, B 0.000, C 0.000 }
gfCNCPoint5[8896] = {X 519.9691, Y 21.6857, Z -7.1667, A 0.000, B 0.000, C 0.000 }
gfCNCPoint5[8897] = {X 518.9900, Y 21.5754, Z -7.1667, A 0.000, B 0.000, C 0.000 }
gfCNCPoint5[8898] = {X 518.0600, Y 21.2500, Z -7.1667, A 0.000, B 0.000, C 0.000 }
gfCNCPoint5[8899] = {X 517.2257, Y 20.7258, Z -7.1667, A 0.000, B 0.000, C 0.000 }
gfCNCPoint5[8900] = {X 516.5290, Y 20.0291, Z -7.1667, A 0.000, B 0.000, C 0.000 }
gfCNCPoint5[8901] = {X 516.0048, Y 19.1948, Z -7.1667, A 0.000, B 0.000, C 0.000 }
gfCNCPoint5[8902] = {X 515.6794, Y 18.2648, Z -7.1667, A 0.000, B 0.000, C 0.000 }
gfCNCPoint5[8903] = {X 515.5691, Y 17.2857, Z -7.1667, A 0.000, B 0.000, C 0.000 }
gfCNCPoint5[8904] = {X 515.5691, Y 10.3077, Z -7.1667, A 0.000, B 0.000, C 0.000 }
gfCNCPoint5[8905] = {X 515.6394, Y 9.5244, Z -7.1667, A 0.000, B 0.000, C 0.000 }
gfCNCPoint5[8906] = {X 515.8480, Y 8.7661, Z -7.1667, A 0.000, B 0.000, C 0.000 }
gfCNCPoint5[8907] = {X 516.1883, Y 8.0570, Z -7.1667, A 0.000, B 0.000, C 0.000 }
gfCNCPoint5[8908] = {X 516.6494, Y 7.4199, Z -7.1667, A 0.000, B 0.000, C 0.000 }
gfCNCPoint5[8909] = {X 516.2872, Y 7.1049, Z -7.1667, A 0.000, B 0.000, C 0.000 }
gfCNCPoint5[8910] = {X 469.2598, Y 7.1049, Z -7.1667, A 0.000, B 0.000, C 0.000 }
gfCNCPoint5[8911] = {X 469.2598, Y 11.9049, Z -7.1667, A 0.000, B 0.000, C 0.000 }
gfCNCPoint5[8912] = {X 469.1140, Y 11.9049, Z -7.1667, A 0.000, B 0.000, C 0.000 }
gfCNCPoint5[8913] = {X 469.1170, Y 12.0428, Z -7.1667, A 0.000, B 0.000, C 0.000 }
gfCNCPoint5[8914] = {X 469.1179, Y 12.1807, Z -7.1667, A 0.000, B 0.000, C 0.000 }
gfCNCPoint5[8915] = {X 469.1883, Y 12.0425, Z -7.1667, A 0.000, B 0.000, C 0.000 }
gfCNCPoint5[8916] = {X 469.2598, Y 11.9049, Z -7.1667, A 0.000, B 0.000, C 0.000 }
gfCNCPoint5[8917] = {X 469.2598, Y 9.5049, Z -7.1667, A 0.000, B 0.000, C 0.000 }
gfCNCPoint5[8918] = {X 466.2077, Y 9.5049, Z -7.1667, A 0.000, B 0.000, C 0.000 }
gfCNCPoint5[8919] = {X 466.5691, Y 10.7169, Z -7.1667, A 0.000, B 0.000, C 0.000 }
gfCNCPoint5[8920] = {X 466.7150, Y 11.9733, Z -7.1667, A 0.000, B 0.000, C 0.000 }
gfCNCPoint5[8921] = {X 466.7172, Y 12.0770, Z -7.1667, A 0.000, B 0.000, C 0.000 }
gfCNCPoint5[8922] = {X 466.7179, Y 12.1806, Z -7.1667, A 0.000, B 0.000, C 0.000 }
gfCNCPoint5[8923] = {X 466.7179, Y 12.9779, Z -7.1667, A 0.000, B 0.000, C 0.000 }
gfCNCPoint5[8924] = {X 466.6192, Y 14.1730, Z -7.1667, A 0.000, B 0.000, C 0.000 }
gfCNCPoint5[8925] = {X 466.3256, Y 15.3355, Z -7.1667, A 0.000, B 0.000, C 0.000 }
gfCNCPoint5[8926] = {X 465.8452, Y 16.4342, Z -7.1667, A 0.000, B 0.000, C 0.000 }
gfCNCPoint5[8927] = {X 465.1910, Y 17.4390, Z -7.1667, A 0.000, B 0.000, C 0.000 }
gfCNCPoint5[8928] = {X 465.1913, Y 25.8869, Z -7.1667, A 0.000, B 0.000, C 0.000 }
gfCNCPoint5[8929] = {X 467.5913, Y 25.8868, Z -7.1667, A 0.000, B 0.000, C 0.000 }
gfCNCPoint5[8930] = {X 467.5919, Y 38.9919, Z -7.1667, A 0.000, B 0.000, C 0.000 }
gfCNCPoint5[8931] = {X 467.6015, Y 39.0069, Z -7.1667, A 0.000, B 0.000, C 0.000 }
gfCNCPoint5[8932] = {X 468.3506, Y 37.9855, Z -7.1667, A 0.000, B 0.000, C 0.000 }
gfCNCPoint5[8933] = {X 469.2267, Y 37.0706, Z -7.1667, A 0.000, B 0.000, C 0.000 }
gfCNCPoint5[8934] = {X 470.2148, Y 36.2780, Z -7.1667, A 0.000, B 0.000, C 0.000 }
gfCNCPoint5[8935] = {X 471.5269, Y 33.7097, Z -7.1667, A 0.000, B 0.000, C 0.000 }
gfCNCPoint5[8936] = {X 470.4793, Y 32.4132, Z -7.1667, A 0.000, B 0.000, C 0.000 }
gfCNCPoint5[8937] = {X 469.5652, Y 31.0194, Z -7.1667, A 0.000, B 0.000, C 0.000 }
gfCNCPoint5[8938] = {X 468.7936, Y 29.5420, Z -7.1667, A 0.000, B 0.000, C 0.000 }
gfCNCPoint5[8939] = {X 468.1721, Y 27.9954, Z -7.1667, A 0.000, B 0.000, C 0.000 }
gfCNCPoint5[8940] = {X 467.7068, Y 26.3949, Z -7.1667, A 0.000, B 0.000, C 0.000 }
gfCNCPoint5[8941] = {X 467.6476, Y 26.1412, Z -7.1667, A 0.000, B 0.000, C 0.000 }
gfCNCPoint5[8942] = {X 467.5913, Y 25.8868, Z -7.1667, A 0.000, B 0.000, C 0.000 }
gfCNCPoint5[8943] = {X 465.1913, Y 25.8869, Z -7.1667, A 0.000, B 0.000, C 0.000 }
gfCNCPoint5[8944] = {X 465.1919, Y 39.7489, Z -7.1667, A 0.000, B 0.000, C 0.000 }
gfCNCPoint5[8945] = {X 465.3910, Y 40.0184, Z -7.1667, A 0.000, B 0.000, C 0.000 }
gfCNCPoint5[8946] = {X 465.5774, Y 40.2966, Z -7.1667, A 0.000, B 0.000, C 0.000 }
gfCNCPoint5[8947] = {X 466.0634, Y 41.1919, Z -7.1667, A 0.000, B 0.000, C 0.000 }
gfCNCPoint5[8948] = {X 466.4196, Y 42.1462, Z -7.1667, A 0.000, B 0.000, C 0.000 }
gfCNCPoint5[8949] = {X 466.6392, Y 43.1408, Z -7.1667, A 0.000, B 0.000, C 0.000 }
gfCNCPoint5[8950] = {X 466.7178, Y 44.1564, Z -7.1667, A 0.000, B 0.000, C 0.000 }
gfCNCPoint5[8951] = {X 466.7179, Y 45.0000, Z -7.1667, A 0.000, B 0.000, C 0.000 }
gfCNCPoint5[8952] = {X 466.7033, Y 45.4609, Z -7.1667, A 0.000, B 0.000, C 0.000 }
gfCNCPoint5[8953] = {X 466.6596, Y 45.9200, Z -7.1667, A 0.000, B 0.000, C 0.000 }
gfCNCPoint5[8954] = {X 468.5433, Y 45.9200, Z -7.1667, A 0.000, B 0.000, C 0.000 }
gfCNCPoint5[8955] = {X 468.4996, Y 45.4609, Z -7.1667, A 0.000, B 0.000, C 0.000 }
gfCNCPoint5[8956] = {X 468.4850, Y 45.0000, Z -7.1667, A 0.000, B 0.000, C 0.000 }
gfCNCPoint5[8957] = {X 468.4850, Y 44.2089, Z -7.1667, A 0.000, B 0.000, C 0.000 }
gfCNCPoint5[8958] = {X 468.5580, Y 43.1798, Z -7.1667, A 0.000, B 0.000, C 0.000 }
gfCNCPoint5[8959] = {X 468.7759, Y 42.1713, Z -7.1667, A 0.000, B 0.000, C 0.000 }
gfCNCPoint5[8960] = {X 469.1341, Y 41.2038, Z -7.1667, A 0.000, B 0.000, C 0.000 }
gfCNCPoint5[8961] = {X 469.6255, Y 40.2966, Z -7.1667, A 0.000, B 0.000, C 0.000 }
gfCNCPoint5[8962] = {X 470.3102, Y 39.3876, Z -7.1667, A 0.000, B 0.000, C 0.000 }
gfCNCPoint5[8963] = {X 471.1282, Y 38.5964, Z -7.1667, A 0.000, B 0.000, C 0.000 }
gfCNCPoint5[8964] = {X 472.0595, Y 37.9424, Z -7.1667, A 0.000, B 0.000, C 0.000 }
gfCNCPoint5[8965] = {X 474.4563, Y 33.2509, Z -7.1667, A 0.000, B 0.000, C 0.000 }
gfCNCPoint5[8966] = {X 473.2242, Y 32.0062, Z -7.1667, A 0.000, B 0.000, C 0.000 }
gfCNCPoint5[8967] = {X 472.1521, Y 30.6212, Z -7.1667, A 0.000, B 0.000, C 0.000 }
gfCNCPoint5[8968] = {X 471.2558, Y 29.1165, Z -7.1667, A 0.000, B 0.000, C 0.000 }
gfCNCPoint5[8969] = {X 470.5487, Y 27.5141, Z -7.1667, A 0.000, B 0.000, C 0.000 }
gfCNCPoint5[8970] = {X 470.0412, Y 25.8379, Z -7.1667, A 0.000, B 0.000, C 0.000 }
gfCNCPoint5[8971] = {X 469.9882, Y 25.6106, Z -7.1667, A 0.000, B 0.000, C 0.000 }
gfCNCPoint5[8972] = {X 469.9378, Y 25.3828, Z -7.1667, A 0.000, B 0.000, C 0.000 }
gfCNCPoint5[8973] = {X 469.6265, Y 23.4874, Z -7.1667, A 0.000, B 0.000, C 0.000 }
gfCNCPoint5[8974] = {X 469.5012, Y 21.5708, Z -7.1667, A 0.000, B 0.000, C 0.000 }
gfCNCPoint5[8975] = {X 469.5630, Y 19.6510, Z -7.1667, A 0.000, B 0.000, C 0.000 }
gfCNCPoint5[8976] = {X 469.8115, Y 17.7464, Z -7.1667, A 0.000, B 0.000, C 0.000 }
gfCNCPoint5[8977] = {X 470.2441, Y 15.8750, Z -7.1667, A 0.000, B 0.000, C 0.000 }
gfCNCPoint5[8978] = {X 470.6909, Y 14.5429, Z -7.1667, A 0.000, B 0.000, C 0.000 }
gfCNCPoint5[8979] = {X 471.2620, Y 13.2592, Z -7.1667, A 0.000, B 0.000, C 0.000 }
gfCNCPoint5[8980] = {X 471.3225, Y 13.1403, Z -7.1667, A 0.000, B 0.000, C 0.000 }
gfCNCPoint5[8981] = {X 471.3840, Y 13.0219, Z -7.1667, A 0.000, B 0.000, C 0.000 }
gfCNCPoint5[8982] = {X 472.1252, Y 11.7667, Z -7.1667, A 0.000, B 0.000, C 0.000 }
gfCNCPoint5[8983] = {X 472.9863, Y 10.5906, Z -7.1667, A 0.000, B 0.000, C 0.000 }
gfCNCPoint5[8984] = {X 473.9589, Y 9.5049, Z -7.1667, A 0.000, B 0.000, C 0.000 }
gfCNCPoint5[8985] = {X 469.2598, Y 9.5049, Z -7.1667, A 0.000, B 0.000, C 0.000 }
gfCNCPoint5[8986] = {X 469.2598, Y 7.1049, Z -7.1667, A 0.000, B 0.000, C 0.000 }
gfCNCPoint5[8987] = {X 370.0985, Y 7.1049, Z -7.1667, A 0.000, B 0.000, C 0.000 }
gfCNCPoint5[8988] = {X 371.1224, Y 8.7924, Z -7.1667, A 0.000, B 0.000, C 0.000 }
gfCNCPoint5[8989] = {X 372.0339, Y 10.5431, Z -7.1667, A 0.000, B 0.000, C 0.000 }
gfCNCPoint5[8990] = {X 372.8310, Y 12.3539, Z -7.1667, A 0.000, B 0.000, C 0.000 }
gfCNCPoint5[8991] = {X 373.5078, Y 14.2131, Z -7.1667, A 0.000, B 0.000, C 0.000 }
gfCNCPoint5[8992] = {X 374.0615, Y 16.1125, Z -7.1667, A 0.000, B 0.000, C 0.000 }
gfCNCPoint5[8993] = {X 374.6275, Y 18.7971, Z -7.1667, A 0.000, B 0.000, C 0.000 }
gfCNCPoint5[8994] = {X 374.9928, Y 21.5163, Z -7.1667, A 0.000, B 0.000, C 0.000 }
gfCNCPoint5[8995] = {X 375.1553, Y 24.2551, Z -7.1667, A 0.000, B 0.000, C 0.000 }
gfCNCPoint5[8996] = {X 375.1141, Y 26.9984, Z -7.1667, A 0.000, B 0.000, C 0.000 }
gfCNCPoint5[8997] = {X 374.8695, Y 29.7311, Z -7.1667, A 0.000, B 0.000, C 0.000 }
gfCNCPoint5[8998] = {X 374.4227, Y 32.4381, Z -7.1667, A 0.000, B 0.000, C 0.000 }
gfCNCPoint5[8999] = {X 373.7849, Y 34.9986, Z -7.1667, A 0.000, B 0.000, C 0.000 }
gfCNCPoint5[9000] = {X 372.9238, Y 37.4928, Z -7.1667, A 0.000, B 0.000, C 0.000 }
gfCNCPoint5[9001] = {X 371.8461, Y 39.9014, Z -7.1667, A 0.000, B 0.000, C 0.000 }
gfCNCPoint5[9002] = {X 370.5602, Y 42.2056, Z -7.1667, A 0.000, B 0.000, C 0.000 }
gfCNCPoint5[9003] = {X 369.0762, Y 44.3874, Z -7.1667, A 0.000, B 0.000, C 0.000 }
gfCNCPoint5[9004] = {X 369.0354, Y 44.4424, Z -7.1667, A 0.000, B 0.000, C 0.000 }
gfCNCPoint5[9005] = {X 368.9945, Y 44.4972, Z -7.1667, A 0.000, B 0.000, C 0.000 }
gfCNCPoint5[9006] = {X 367.5951, Y 46.2173, Z -7.1667, A 0.000, B 0.000, C 0.000 }
gfCNCPoint5[9007] = {X 366.0610, Y 47.8183, Z -7.1667, A 0.000, B 0.000, C 0.000 }
gfCNCPoint5[9008] = {X 364.4022, Y 49.2898, Z -7.1667, A 0.000, B 0.000, C 0.000 }
gfCNCPoint5[9009] = {X 362.6297, Y 50.6220, Z -7.1667, A 0.000, B 0.000, C 0.000 }
gfCNCPoint5[9010] = {X 360.7550, Y 51.8062, Z -7.1667, A 0.000, B 0.000, C 0.000 }
gfCNCPoint5[9011] = {X 358.7906, Y 52.8347, Z -7.1667, A 0.000, B 0.000, C 0.000 }
gfCNCPoint5[9012] = {X 358.6058, Y 52.9212, Z -7.1667, A 0.000, B 0.000, C 0.000 }
gfCNCPoint5[9013] = {X 358.4204, Y 53.0064, Z -7.1667, A 0.000, B 0.000, C 0.000 }
gfCNCPoint5[9014] = {X 356.1469, Y 53.8831, Z -7.1667, A 0.000, B 0.000, C 0.000 }
gfCNCPoint5[9015] = {X 353.8067, Y 54.5615, Z -7.1667, A 0.000, B 0.000, C 0.000 }
gfCNCPoint5[9016] = {X 351.4168, Y 55.0368, Z -7.1667, A 0.000, B 0.000, C 0.000 }
gfCNCPoint5[9017] = {X 348.9950, Y 55.3053, Z -7.1667, A 0.000, B 0.000, C 0.000 }
gfCNCPoint5[9018] = {X 349.9663, Y 69.6725, Z -7.1667, A 0.000, B 0.000, C 0.000 }
gfCNCPoint5[9019] = {X 348.6649, Y 69.7406, Z -7.1667, A 0.000, B 0.000, C 0.000 }
gfCNCPoint5[9020] = {X 347.3621, Y 69.7690, Z -7.1667, A 0.000, B 0.000, C 0.000 }
gfCNCPoint5[9021] = {X 346.5845, Y 69.7781, Z -7.1667, A 0.000, B 0.000, C 0.000 }
gfCNCPoint5[9022] = {X 345.8069, Y 69.7734, Z -7.1667, A 0.000, B 0.000, C 0.000 }
gfCNCPoint5[9023] = {X 345.5915, Y 70.1904, Z -7.1667, A 0.000, B 0.000, C 0.000 }
gfCNCPoint5[9024] = {X 345.3680, Y 70.6031, Z -7.1667, A 0.000, B 0.000, C 0.000 }
gfCNCPoint5[9025] = {X 347.2080, Y 70.6204, Z -7.1667, A 0.000, B 0.000, C 0.000 }
gfCNCPoint5[9026] = {X 349.0480, Y 70.6087, Z -7.1667, A 0.000, B 0.000, C 0.000 }
gfCNCPoint5[9027] = {X 349.7517, Y 70.6084, Z -7.1667, A 0.000, B 0.000, C 0.000 }
gfCNCPoint5[9028] = {X 350.4554, Y 70.6029, Z -7.1667, A 0.000, B 0.000, C 0.000 }
gfCNCPoint5[9029] = {X 350.2058, Y 70.1404, Z -7.1667, A 0.000, B 0.000, C 0.000 }
gfCNCPoint5[9030] = {X 349.9663, Y 69.6725, Z -7.1667, A 0.000, B 0.000, C 0.000 }
gfCNCPoint5[9031] = {X 349.8044, Y 67.2780, Z -7.1667, A 0.000, B 0.000, C 0.000 }
gfCNCPoint5[9032] = {X 348.5676, Y 67.3425, Z -7.1667, A 0.000, B 0.000, C 0.000 }
gfCNCPoint5[9033] = {X 347.3294, Y 67.3692, Z -7.1667, A 0.000, B 0.000, C 0.000 }
gfCNCPoint5[9034] = {X 345.8127, Y 67.3732, Z -7.1667, A 0.000, B 0.000, C 0.000 }
gfCNCPoint5[9035] = {X 344.2968, Y 67.3214, Z -7.1667, A 0.000, B 0.000, C 0.000 }
gfCNCPoint5[9036] = {X 343.8116, Y 68.3945, Z -7.1667, A 0.000, B 0.000, C 0.000 }
gfCNCPoint5[9037] = {X 343.2688, Y 69.4398, Z -7.1667, A 0.000, B 0.000, C 0.000 }
gfCNCPoint5[9038] = {X 342.7888, Y 70.2629, Z -7.1667, A 0.000, B 0.000, C 0.000 }
gfCNCPoint5[9039] = {X 342.2731, Y 71.0641, Z -7.1667, A 0.000, B 0.000, C 0.000 }
gfCNCPoint5[9040] = {X 342.2733, Y 72.9108, Z -7.1667, A 0.000, B 0.000, C 0.000 }
gfCNCPoint5[9041] = {X 343.7996, Y 72.9666, Z -7.1667, A 0.000, B 0.000, C 0.000 }
gfCNCPoint5[9042] = {X 345.3265, Y 73.0028, Z -7.1667, A 0.000, B 0.000, C 0.000 }
gfCNCPoint5[9043] = {X 347.1938, Y 73.0204, Z -7.1667, A 0.000, B 0.000, C 0.000 }
gfCNCPoint5[9044] = {X 349.0612, Y 73.0088, Z -7.1667, A 0.000, B 0.000, C 0.000 }
gfCNCPoint5[9045] = {X 349.7723, Y 73.0084, Z -7.1667, A 0.000, B 0.000, C 0.000 }
gfCNCPoint5[9046] = {X 350.4833, Y 73.0027, Z -7.1667, A 0.000, B 0.000, C 0.000 }
gfCNCPoint5[9047] = {X 352.0212, Y 72.9726, Z -7.1667, A 0.000, B 0.000, C 0.000 }
gfCNCPoint5[9048] = {X 353.5584, Y 72.9182, Z -7.1667, A 0.000, B 0.000, C 0.000 }
gfCNCPoint5[9049] = {X 353.5583, Y 71.0760, Z -7.1667, A 0.000, B 0.000, C 0.000 }
gfCNCPoint5[9050] = {X 353.0385, Y 70.2691, Z -7.1667, A 0.000, B 0.000, C 0.000 }
gfCNCPoint5[9051] = {X 352.5548, Y 69.4399, Z -7.1667, A 0.000, B 0.000, C 0.000 }
gfCNCPoint5[9052] = {X 351.9680, Y 68.3027, Z -7.1667, A 0.000, B 0.000, C 0.000 }
gfCNCPoint5[9053] = {X 351.4494, Y 67.1329, Z -7.1667, A 0.000, B 0.000, C 0.000 }
gfCNCPoint5[9054] = {X 350.6276, Y 67.2139, Z -7.1667, A 0.000, B 0.000, C 0.000 }
gfCNCPoint5[9055] = {X 349.8044, Y 67.2780, Z -7.1667, A 0.000, B 0.000, C 0.000 }
gfCNCPoint5[9056] = {X 349.6425, Y 64.8834, Z -7.1667, A 0.000, B 0.000, C 0.000 }
gfCNCPoint5[9057] = {X 348.4703, Y 64.9445, Z -7.1667, A 0.000, B 0.000, C 0.000 }
gfCNCPoint5[9058] = {X 347.2967, Y 64.9693, Z -7.1667, A 0.000, B 0.000, C 0.000 }
gfCNCPoint5[9059] = {X 344.9827, Y 64.9501, Z -7.1667, A 0.000, B 0.000, C 0.000 }
gfCNCPoint5[9060] = {X 342.6740, Y 64.7929, Z -7.1667, A 0.000, B 0.000, C 0.000 }
gfCNCPoint5[9061] = {X 341.9395, Y 66.7274, Z -7.1667, A 0.000, B 0.000, C 0.000 }
gfCNCPoint5[9062] = {X 341.0022, Y 68.5723, Z -7.1667, A 0.000, B 0.000, C 0.000 }
gfCNCPoint5[9063] = {X 339.8730, Y 70.3063, Z -7.1667, A 0.000, B 0.000, C 0.000 }
gfCNCPoint5[9064] = {X 339.8735, Y 75.1881, Z -7.1667, A 0.000, B 0.000, C 0.000 }
gfCNCPoint5[9065] = {X 344.4719, Y 75.3856, Z -7.1667, A 0.000, B 0.000, C 0.000 }
gfCNCPoint5[9066] = {X 349.0745, Y 75.4088, Z -7.1667, A 0.000, B 0.000, C 0.000 }
gfCNCPoint5[9067] = {X 352.5184, Y 75.3590, Z -7.1667, A 0.000, B 0.000, C 0.000 }
gfCNCPoint5[9068] = {X 355.9586, Y 75.1898, Z -7.1667, A 0.000, B 0.000, C 0.000 }
gfCNCPoint5[9069] = {X 355.9583, Y 70.3171, Z -7.1667, A 0.000, B 0.000, C 0.000 }
gfCNCPoint5[9070] = {X 355.0508, Y 68.9595, Z -7.1667, A 0.000, B 0.000, C 0.000 }
gfCNCPoint5[9071] = {X 354.2615, Y 67.5299, Z -7.1667, A 0.000, B 0.000, C 0.000 }
gfCNCPoint5[9072] = {X 353.5960, Y 66.0387, Z -7.1667, A 0.000, B 0.000, C 0.000 }
gfCNCPoint5[9073] = {X 353.0591, Y 64.4965, Z -7.1667, A 0.000, B 0.000, C 0.000 }
gfCNCPoint5[9074] = {X 351.3552, Y 64.7286, Z -7.1667, A 0.000, B 0.000, C 0.000 }
gfCNCPoint5[9075] = {X 349.6425, Y 64.8834, Z -7.1667, A 0.000, B 0.000, C 0.000 }
gfCNCPoint5[9076] = {X 349.4807, Y 62.4889, Z -7.1667, A 0.000, B 0.000, C 0.000 }
gfCNCPoint5[9077] = {X 348.3730, Y 62.5464, Z -7.1667, A 0.000, B 0.000, C 0.000 }
gfCNCPoint5[9078] = {X 347.2640, Y 62.5694, Z -7.1667, A 0.000, B 0.000, C 0.000 }
gfCNCPoint5[9079] = {X 345.1285, Y 62.5539, Z -7.1667, A 0.000, B 0.000, C 0.000 }
gfCNCPoint5[9080] = {X 342.9976, Y 62.4130, Z -7.1667, A 0.000, B 0.000, C 0.000 }
gfCNCPoint5[9081] = {X 340.8786, Y 62.1473, Z -7.1667, A 0.000, B 0.000, C 0.000 }
gfCNCPoint5[9082] = {X 340.4889, Y 63.7350, Z -7.1667, A 0.000, B 0.000, C 0.000 }
gfCNCPoint5[9083] = {X 339.9477, Y 65.2777, Z -7.1667, A 0.000, B 0.000, C 0.000 }
gfCNCPoint5[9084] = {X 339.2602, Y 66.7609, Z -7.1667, A 0.000, B 0.000, C 0.000 }
gfCNCPoint5[9085] = {X 338.4327, Y 68.1708, Z -7.1667, A 0.000, B 0.000, C 0.000 }
gfCNCPoint5[9086] = {X 337.4729, Y 69.4943, Z -7.1667, A 0.000, B 0.000, C 0.000 }
gfCNCPoint5[9087] = {X 337.4737, Y 77.4234, Z -7.1667, A 0.000, B 0.000, C 0.000 }
gfCNCPoint5[9088] = {X 341.3404, Y 77.6730, Z -7.1667, A 0.000, B 0.000, C 0.000 }
gfCNCPoint5[9089] = {X 345.2130, Y 77.8015, Z -7.1667, A 0.000, B 0.000, C 0.000 }
gfCNCPoint5[9090] = {X 349.0878, Y 77.8089, Z -7.1667, A 0.000, B 0.000, C 0.000 }
gfCNCPoint5[9091] = {X 353.7278, Y 77.7154, Z -7.1667, A 0.000, B 0.000, C 0.000 }
gfCNCPoint5[9092] = {X 358.3587, Y 77.4104, Z -7.1667, A 0.000, B 0.000, C 0.000 }
gfCNCPoint5[9093] = {X 358.3582, Y 69.5039, Z -7.1667, A 0.000, B 0.000, C 0.000 }
gfCNCPoint5[9094] = {X 357.3475, Y 68.1043, Z -7.1667, A 0.000, B 0.000, C 0.000 }
gfCNCPoint5[9095] = {X 356.4849, Y 66.6088, Z -7.1667, A 0.000, B 0.000, C 0.000 }
gfCNCPoint5[9096] = {X 355.7796, Y 65.0330, Z -7.1667, A 0.000, B 0.000, C 0.000 }
gfCNCPoint5[9097] = {X 355.2390, Y 63.3935, Z -7.1667, A 0.000, B 0.000, C 0.000 }
gfCNCPoint5[9098] = {X 354.8686, Y 61.7072, Z -7.1667, A 0.000, B 0.000, C 0.000 }
gfCNCPoint5[9099] = {X 352.1896, Y 62.2013, Z -7.1667, A 0.000, B 0.000, C 0.000 }
gfCNCPoint5[9100] = {X 349.4807, Y 62.4889, Z -7.1667, A 0.000, B 0.000, C 0.000 }
gfCNCPoint5[9101] = {X 349.3188, Y 60.0944, Z -7.1667, A 0.000, B 0.000, C 0.000 }
gfCNCPoint5[9102] = {X 348.2756, Y 60.1484, Z -7.1667, A 0.000, B 0.000, C 0.000 }
gfCNCPoint5[9103] = {X 347.2313, Y 60.1696, Z -7.1667, A 0.000, B 0.000, C 0.000 }
gfCNCPoint5[9104] = {X 344.3951, Y 60.1154, Z -7.1667, A 0.000, B 0.000, C 0.000 }
gfCNCPoint5[9105] = {X 341.5733, Y 59.8248, Z -7.1667, A 0.000, B 0.000, C 0.000 }
gfCNCPoint5[9106] = {X 338.7856, Y 59.2998, Z -7.1667, A 0.000, B 0.000, C 0.000 }
gfCNCPoint5[9107] = {X 338.6401, Y 60.9990, Z -7.1667, A 0.000, B 0.000, C 0.000 }
gfCNCPoint5[9108] = {X 338.2963, Y 62.6694, Z -7.1667, A 0.000, B 0.000, C 0.000 }
gfCNCPoint5[9109] = {X 337.7590, Y 64.2879, Z -7.1667, A 0.000, B 0.000, C 0.000 }
gfCNCPoint5[9110] = {X 337.0356, Y 65.8323, Z -7.1667, A 0.000, B 0.000, C 0.000 }
gfCNCPoint5[9111] = {X 336.1361, Y 67.2812, Z -7.1667, A 0.000, B 0.000, C 0.000 }
gfCNCPoint5[9112] = {X 335.0728, Y 68.6146, Z -7.1667, A 0.000, B 0.000, C 0.000 }
gfCNCPoint5[9113] = {X 335.0739, Y 79.5854, Z -7.1667, A 0.000, B 0.000, C 0.000 }
gfCNCPoint5[9114] = {X 335.9840, Y 79.6949, Z -7.1667, A 0.000, B 0.000, C 0.000 }
gfCNCPoint5[9115] = {X 336.8962, Y 79.7841, Z -7.1667, A 0.000, B 0.000, C 0.000 }
gfCNCPoint5[9116] = {X 340.9593, Y 80.0569, Z -7.1667, A 0.000, B 0.000, C 0.000 }
gfCNCPoint5[9117] = {X 345.0290, Y 80.1986, Z -7.1667, A 0.000, B 0.000, C 0.000 }
gfCNCPoint5[9118] = {X 349.1011, Y 80.2089, Z -7.1667, A 0.000, B 0.000, C 0.000 }
gfCNCPoint5[9119] = {X 352.9063, Y 80.1488, Z -7.1667, A 0.000, B 0.000, C 0.000 }
gfCNCPoint5[9120] = {X 356.7068, Y 79.9497, Z -7.1667, A 0.000, B 0.000, C 0.000 }
gfCNCPoint5[9121] = {X 360.4975, Y 79.6119, Z -7.1667, A 0.000, B 0.000, C 0.000 }
gfCNCPoint5[9122] = {X 360.7588, Y 79.5819, Z -7.1667, A 0.000, B 0.000, C 0.000 }
gfCNCPoint5[9123] = {X 360.7582, Y 68.6227, Z -7.1667, A 0.000, B 0.000, C 0.000 }
gfCNCPoint5[9124] = {X 359.7293, Y 67.3405, Z -7.1667, A 0.000, B 0.000, C 0.000 }
gfCNCPoint5[9125] = {X 358.8525, Y 65.9499, Z -7.1667, A 0.000, B 0.000, C 0.000 }
gfCNCPoint5[9126] = {X 358.1389, Y 64.4689, Z -7.1667, A 0.000, B 0.000, C 0.000 }
gfCNCPoint5[9127] = {X 357.5977, Y 62.9166, Z -7.1667, A 0.000, B 0.000, C 0.000 }
gfCNCPoint5[9128] = {X 357.2360, Y 61.3129, Z -7.1667, A 0.000, B 0.000, C 0.000 }
gfCNCPoint5[9129] = {X 357.0916, Y 60.1641, Z -7.1667, A 0.000, B 0.000, C 0.000 }
gfCNCPoint5[9130] = {X 357.0395, Y 59.0073, Z -7.1667, A 0.000, B 0.000, C 0.000 }
gfCNCPoint5[9131] = {X 357.0394, Y 58.6404, Z -7.1667, A 0.000, B 0.000, C 0.000 }
gfCNCPoint5[9132] = {X 355.6990, Y 59.0313, Z -7.1667, A 0.000, B 0.000, C 0.000 }
gfCNCPoint5[9133] = {X 354.3434, Y 59.3654, Z -7.1667, A 0.000, B 0.000, C 0.000 }
gfCNCPoint5[9134] = {X 351.8450, Y 59.8261, Z -7.1667, A 0.000, B 0.000, C 0.000 }
gfCNCPoint5[9135] = {X 349.3188, Y 60.0944, Z -7.1667, A 0.000, B 0.000, C 0.000 }
gfCNCPoint5[9136] = {X 349.1569, Y 57.6998, Z -7.1667, A 0.000, B 0.000, C 0.000 }
gfCNCPoint5[9137] = {X 348.1784, Y 57.7503, Z -7.1667, A 0.000, B 0.000, C 0.000 }
gfCNCPoint5[9138] = {X 347.1987, Y 57.7697, Z -7.1667, A 0.000, B 0.000, C 0.000 }
gfCNCPoint5[9139] = {X 344.5556, Y 57.7208, Z -7.1667, A 0.000, B 0.000, C 0.000 }
gfCNCPoint5[9140] = {X 341.9258, Y 57.4508, Z -7.1667, A 0.000, B 0.000, C 0.000 }
gfCNCPoint5[9141] = {X 339.3279, Y 56.9619, Z -7.1667, A 0.000, B 0.000, C 0.000 }
gfCNCPoint5[9142] = {X 337.7710, Y 56.5587, Z -7.1667, A 0.000, B 0.000, C 0.000 }
gfCNCPoint5[9143] = {X 336.2366, Y 56.0767, Z -7.1667, A 0.000, B 0.000, C 0.000 }
gfCNCPoint5[9144] = {X 336.3521, Y 57.0353, Z -7.1667, A 0.000, B 0.000, C 0.000 }
gfCNCPoint5[9145] = {X 336.3907, Y 58.0000, Z -7.1667, A 0.000, B 0.000, C 0.000 }
gfCNCPoint5[9146] = {X 336.3907, Y 58.9512, Z -7.1667, A 0.000, B 0.000, C 0.000 }
gfCNCPoint5[9147] = {X 336.3894, Y 59.0935, Z -7.1667, A 0.000, B 0.000, C 0.000 }
gfCNCPoint5[9148] = {X 336.3864, Y 59.2358, Z -7.1667, A 0.000, B 0.000, C 0.000 }
gfCNCPoint5[9149] = {X 336.2429, Y 60.7999, Z -7.1667, A 0.000, B 0.000, C 0.000 }
gfCNCPoint5[9150] = {X 335.8983, Y 62.3322, Z -7.1667, A 0.000, B 0.000, C 0.000 }
gfCNCPoint5[9151] = {X 335.3583, Y 63.8071, Z -7.1667, A 0.000, B 0.000, C 0.000 }
gfCNCPoint5[9152] = {X 334.6321, Y 65.1998, Z -7.1667, A 0.000, B 0.000, C 0.000 }
gfCNCPoint5[9153] = {X 333.7319, Y 66.4869, Z -7.1667, A 0.000, B 0.000, C 0.000 }
gfCNCPoint5[9154] = {X 332.6728, Y 67.6467, Z -7.1667, A 0.000, B 0.000, C 0.000 }
gfCNCPoint5[9155] = {X 332.6741, Y 81.6388, Z -7.1667, A 0.000, B 0.000, C 0.000 }
gfCNCPoint5[9156] = {X 334.6773, Y 81.9539, Z -7.1667, A 0.000, B 0.000, C 0.000 }
gfCNCPoint5[9157] = {X 336.6931, Y 82.1755, Z -7.1667, A 0.000, B 0.000, C 0.000 }
gfCNCPoint5[9158] = {X 340.8282, Y 82.4534, Z -7.1667, A 0.000, B 0.000, C 0.000 }
gfCNCPoint5[9159] = {X 344.9701, Y 82.5979, Z -7.1667, A 0.000, B 0.000, C 0.000 }
gfCNCPoint5[9160] = {X 349.1145, Y 82.6090, Z -7.1667, A 0.000, B 0.000, C 0.000 }
gfCNCPoint5[9161] = {X 353.0020, Y 82.5469, Z -7.1667, A 0.000, B 0.000, C 0.000 }
gfCNCPoint5[9162] = {X 356.8846, Y 82.3431, Z -7.1667, A 0.000, B 0.000, C 0.000 }
gfCNCPoint5[9163] = {X 360.7571, Y 81.9979, Z -7.1667, A 0.000, B 0.000, C 0.000 }
gfCNCPoint5[9164] = {X 361.9617, Y 81.8407, Z -7.1667, A 0.000, B 0.000, C 0.000 }
gfCNCPoint5[9165] = {X 363.1589, Y 81.6351, Z -7.1667, A 0.000, B 0.000, C 0.000 }
gfCNCPoint5[9166] = {X 363.1581, Y 67.6529, Z -7.1667, A 0.000, B 0.000, C 0.000 }
gfCNCPoint5[9167] = {X 362.0722, Y 66.4627, Z -7.1667, A 0.000, B 0.000, C 0.000 }
gfCNCPoint5[9168] = {X 361.1544, Y 65.1385, Z -7.1667, A 0.000, B 0.000, C 0.000 }
gfCNCPoint5[9169] = {X 360.4209, Y 63.7040, Z -7.1667, A 0.000, B 0.000, C 0.000 }
gfCNCPoint5[9170] = {X 359.8848, Y 62.1846, Z -7.1667, A 0.000, B 0.000, C 0.000 }
gfCNCPoint5[9171] = {X 359.5557, Y 60.6075, Z -7.1667, A 0.000, B 0.000, C 0.000 }
gfCNCPoint5[9172] = {X 359.4395, Y 59.0005, Z -7.1667, A 0.000, B 0.000, C 0.000 }
gfCNCPoint5[9173] = {X 359.4393, Y 58.0000, Z -7.1667, A 0.000, B 0.000, C 0.000 }
gfCNCPoint5[9174] = {X 359.5340, Y 56.4903, Z -7.1667, A 0.000, B 0.000, C 0.000 }
gfCNCPoint5[9175] = {X 359.8166, Y 55.0043, Z -7.1667, A 0.000, B 0.000, C 0.000 }
gfCNCPoint5[9176] = {X 359.6070, Y 55.1025, Z -7.1667, A 0.000, B 0.000, C 0.000 }
gfCNCPoint5[9177] = {X 359.3966, Y 55.1990, Z -7.1667, A 0.000, B 0.000, C 0.000 }
gfCNCPoint5[9178] = {X 357.8733, Y 55.8161, Z -7.1667, A 0.000, B 0.000, C 0.000 }
gfCNCPoint5[9179] = {X 356.3192, Y 56.3510, Z -7.1667, A 0.000, B 0.000, C 0.000 }
gfCNCPoint5[9180] = {X 353.9698, Y 56.9892, Z -7.1667, A 0.000, B 0.000, C 0.000 }
gfCNCPoint5[9181] = {X 351.5774, Y 57.4397, Z -7.1667, A 0.000, B 0.000, C 0.000 }
gfCNCPoint5[9182] = {X 349.1569, Y 57.6998, Z -7.1667, A 0.000, B 0.000, C 0.000 }
gfCNCPoint5[9183] = {X 348.9950, Y 55.3053, Z -7.1667, A 0.000, B 0.000, C 0.000 }
gfCNCPoint5[9184] = {X 348.0811, Y 55.3523, Z -7.1667, A 0.000, B 0.000, C 0.000 }
gfCNCPoint5[9185] = {X 347.1660, Y 55.3698, Z -7.1667, A 0.000, B 0.000, C 0.000 }
gfCNCPoint5[9186] = {X 344.5860, Y 55.3180, Z -7.1667, A 0.000, B 0.000, C 0.000 }
gfCNCPoint5[9187] = {X 342.0206, Y 55.0383, Z -7.1667, A 0.000, B 0.000, C 0.000 }
gfCNCPoint5[9188] = {X 339.4900, Y 54.5330, Z -7.1667, A 0.000, B 0.000, C 0.000 }
gfCNCPoint5[9189] = {X 337.0139, Y 53.8061, Z -7.1667, A 0.000, B 0.000, C 0.000 }
gfCNCPoint5[9190] = {X 334.7571, Y 52.9272, Z -7.1667, A 0.000, B 0.000, C 0.000 }
gfCNCPoint5[9191] = {X 332.5810, Y 51.8642, Z -7.1667, A 0.000, B 0.000, C 0.000 }
gfCNCPoint5[9192] = {X 331.5868, Y 51.2792, Z -7.1667, A 0.000, B 0.000, C 0.000 }
gfCNCPoint5[9193] = {X 330.6163, Y 50.6555, Z -7.1667, A 0.000, B 0.000, C 0.000 }
gfCNCPoint5[9194] = {X 331.5814, Y 51.6094, Z -7.1667, A 0.000, B 0.000, C 0.000 }
gfCNCPoint5[9195] = {X 332.4035, Y 52.6889, Z -7.1667, A 0.000, B 0.000, C 0.000 }
gfCNCPoint5[9196] = {X 333.0667, Y 53.8727, Z -7.1667, A 0.000, B 0.000, C 0.000 }
gfCNCPoint5[9197] = {X 333.5578, Y 55.1376, Z -7.1667, A 0.000, B 0.000, C 0.000 }
gfCNCPoint5[9198] = {X 333.8672, Y 56.4588, Z -7.1667, A 0.000, B 0.000, C 0.000 }
gfCNCPoint5[9199] = {X 333.9598, Y 57.2269, Z -7.1667, A 0.000, B 0.000, C 0.000 }
gfCNCPoint5[9200] = {X 333.9907, Y 58.0000, Z -7.1667, A 0.000, B 0.000, C 0.000 }
gfCNCPoint5[9201] = {X 333.9907, Y 58.9436, Z -7.1667, A 0.000, B 0.000, C 0.000 }
gfCNCPoint5[9202] = {X 333.8764, Y 60.3990, Z -7.1667, A 0.000, B 0.000, C 0.000 }
gfCNCPoint5[9203] = {X 333.5454, Y 61.8208, Z -7.1667, A 0.000, B 0.000, C 0.000 }
gfCNCPoint5[9204] = {X 333.0052, Y 63.1769, Z -7.1667, A 0.000, B 0.000, C 0.000 }
gfCNCPoint5[9205] = {X 332.2678, Y 64.4369, Z -7.1667, A 0.000, B 0.000, C 0.000 }
gfCNCPoint5[9206] = {X 331.3501, Y 65.5721, Z -7.1667, A 0.000, B 0.000, C 0.000 }
gfCNCPoint5[9207] = {X 330.2726, Y 66.5571, Z -7.1667, A 0.000, B 0.000, C 0.000 }
gfCNCPoint5[9208] = {X 330.2742, Y 83.2031, Z -7.1667, A 0.000, B 0.000, C 0.000 }
gfCNCPoint5[9209] = {X 330.2780, Y 83.5899, Z -7.1667, A 0.000, B 0.000, C 0.000 }
gfCNCPoint5[9210] = {X 330.5994, Y 83.6703, Z -7.1667, A 0.000, B 0.000, C 0.000 }
gfCNCPoint5[9211] = {X 330.9232, Y 83.7405, Z -7.1667, A 0.000, B 0.000, C 0.000 }
gfCNCPoint5[9212] = {X 333.6939, Y 84.2389, Z -7.1667, A 0.000, B 0.000, C 0.000 }
gfCNCPoint5[9213] = {X 336.4899, Y 84.5669, Z -7.1667, A 0.000, B 0.000, C 0.000 }
gfCNCPoint5[9214] = {X 340.6971, Y 84.8498, Z -7.1667, A 0.000, B 0.000, C 0.000 }
gfCNCPoint5[9215] = {X 344.9113, Y 84.9972, Z -7.1667, A 0.000, B 0.000, C 0.000 }
gfCNCPoint5[9216] = {X 349.1279, Y 85.0090, Z -7.1667, A 0.000, B 0.000, C 0.000 }
gfCNCPoint5[9217] = {X 353.0976, Y 84.9450, Z -7.1667, A 0.000, B 0.000, C 0.000 }
gfCNCPoint5[9218] = {X 357.0623, Y 84.7365, Z -7.1667, A 0.000, B 0.000, C 0.000 }
gfCNCPoint5[9219] = {X 361.0167, Y 84.3838, Z -7.1667, A 0.000, B 0.000, C 0.000 }
gfCNCPoint5[9220] = {X 363.3026, Y 84.0499, Z -7.1667, A 0.000, B 0.000, C 0.000 }
gfCNCPoint5[9221] = {X 365.5591, Y 83.5547, Z -7.1667, A 0.000, B 0.000, C 0.000 }
gfCNCPoint5[9222] = {X 365.5581, Y 66.5608, Z -7.1667, A 0.000, B 0.000, C 0.000 }
gfCNCPoint5[9223] = {X 364.4839, Y 65.5828, Z -7.1667, A 0.000, B 0.000, C 0.000 }
gfCNCPoint5[9224] = {X 363.5681, Y 64.4551, Z -7.1667, A 0.000, B 0.000, C 0.000 }
gfCNCPoint5[9225] = {X 362.8315, Y 63.2030, Z -7.1667, A 0.000, B 0.000, C 0.000 }
gfCNCPoint5[9226] = {X 362.2904, Y 61.8549, Z -7.1667, A 0.000, B 0.000, C 0.000 }
gfCNCPoint5[9227] = {X 361.9573, Y 60.4409, Z -7.1667, A 0.000, B 0.000, C 0.000 }
gfCNCPoint5[9228] = {X 361.8395, Y 58.9930, Z -7.1667, A 0.000, B 0.000, C 0.000 }
gfCNCPoint5[9229] = {X 361.8393, Y 58.0000, Z -7.1667, A 0.000, B 0.000, C 0.000 }
gfCNCPoint5[9230] = {X 361.9152, Y 56.7903, Z -7.1667, A 0.000, B 0.000, C 0.000 }
gfCNCPoint5[9231] = {X 362.1417, Y 55.5995, Z -7.1667, A 0.000, B 0.000, C 0.000 }
gfCNCPoint5[9232] = {X 362.5726, Y 54.3042, Z -7.1667, A 0.000, B 0.000, C 0.000 }
gfCNCPoint5[9233] = {X 363.1814, Y 53.0824, Z -7.1667, A 0.000, B 0.000, C 0.000 }
gfCNCPoint5[9234] = {X 363.9561, Y 51.9584, Z -7.1667, A 0.000, B 0.000, C 0.000 }
gfCNCPoint5[9235] = {X 364.8811, Y 50.9546, Z -7.1667, A 0.000, B 0.000, C 0.000 }
gfCNCPoint5[9236] = {X 365.9382, Y 50.0909, Z -7.1667, A 0.000, B 0.000, C 0.000 }
gfCNCPoint5[9237] = {X 367.1063, Y 49.3844, Z -7.1667, A 0.000, B 0.000, C 0.000 }
gfCNCPoint5[9238] = {X 368.3621, Y 48.8493, Z -7.1667, A 0.000, B 0.000, C 0.000 }
gfCNCPoint5[9239] = {X 369.6807, Y 48.4962, Z -7.1667, A 0.000, B 0.000, C 0.000 }
gfCNCPoint5[9240] = {X 371.0359, Y 48.3321, Z -7.1667, A 0.000, B 0.000, C 0.000 }
gfCNCPoint5[9241] = {X 371.2775, Y 48.3230, Z -7.1667, A 0.000, B 0.000, C 0.000 }
gfCNCPoint5[9242] = {X 371.5193, Y 48.3200, Z -7.1667, A 0.000, B 0.000, C 0.000 }
gfCNCPoint5[9243] = {X 388.0597, Y 48.3200, Z -7.1667, A 0.000, B 0.000, C 0.000 }
gfCNCPoint5[9244] = {X 389.4419, Y 48.4192, Z -7.1667, A 0.000, B 0.000, C 0.000 }
gfCNCPoint5[9245] = {X 390.7958, Y 48.7147, Z -7.1667, A 0.000, B 0.000, C 0.000 }
gfCNCPoint5[9246] = {X 392.0936, Y 49.2006, Z -7.1667, A 0.000, B 0.000, C 0.000 }
gfCNCPoint5[9247] = {X 393.3087, Y 49.8667, Z -7.1667, A 0.000, B 0.000, C 0.000 }
gfCNCPoint5[9248] = {X 394.5333, Y 49.1962, Z -7.1667, A 0.000, B 0.000, C 0.000 }
gfCNCPoint5[9249] = {X 395.8416, Y 48.7089, Z -7.1667, A 0.000, B 0.000, C 0.000 }
gfCNCPoint5[9250] = {X 397.1858, Y 48.4177, Z -7.1667, A 0.000, B 0.000, C 0.000 }
gfCNCPoint5[9251] = {X 398.5577, Y 48.3200, Z -7.1667, A 0.000, B 0.000, C 0.000 }
gfCNCPoint5[9252] = {X 398.7346, Y 48.3200, Z -7.1667, A 0.000, B 0.000, C 0.000 }
gfCNCPoint5[9253] = {X 398.1859, Y 47.6069, Z -7.1667, A 0.000, B 0.000, C 0.000 }
gfCNCPoint5[9254] = {X 397.7774, Y 46.8051, Z -7.1667, A 0.000, B 0.000, C 0.000 }
gfCNCPoint5[9255] = {X 397.5230, Y 45.9420, Z -7.1667, A 0.000, B 0.000, C 0.000 }
gfCNCPoint5[9256] = {X 397.4561, Y 45.4921, Z -7.1667, A 0.000, B 0.000, C 0.000 }
gfCNCPoint5[9257] = {X 397.4314, Y 45.0378, Z -7.1667, A 0.000, B 0.000, C 0.000 }
gfCNCPoint5[9258] = {X 397.4316, Y 44.1456, Z -7.1667, A 0.000, B 0.000, C 0.000 }
gfCNCPoint5[9259] = {X 397.5413, Y 43.1780, Z -7.1667, A 0.000, B 0.000, C 0.000 }
gfCNCPoint5[9260] = {X 397.8410, Y 42.2514, Z -7.1667, A 0.000, B 0.000, C 0.000 }
gfCNCPoint5[9261] = {X 398.3186, Y 41.4029, Z -7.1667, A 0.000, B 0.000, C 0.000 }
gfCNCPoint5[9262] = {X 398.9552, Y 40.6660, Z -7.1667, A 0.000, B 0.000, C 0.000 }
gfCNCPoint5[9263] = {X 398.9552, Y 31.8254, Z -7.1667, A 0.000, B 0.000, C 0.000 }
gfCNCPoint5[9264] = {X 396.7508, Y 27.9920, Z -7.1667, A 0.000, B 0.000, C 0.000 }
gfCNCPoint5[9265] = {X 386.3481, Y 33.9740, Z -7.1667, A 0.000, B 0.000, C 0.000 }
gfCNCPoint5[9266] = {X 386.2673, Y 34.4005, Z -7.1667, A 0.000, B 0.000, C 0.000 }
gfCNCPoint5[9267] = {X 386.1827, Y 34.8263, Z -7.1667, A 0.000, B 0.000, C 0.000 }
gfCNCPoint5[9268] = {X 386.0238, Y 35.5746, Z -7.1667, A 0.000, B 0.000, C 0.000 }
gfCNCPoint5[9269] = {X 385.8513, Y 36.3200, Z -7.1667, A 0.000, B 0.000, C 0.000 }
gfCNCPoint5[9270] = {X 386.9552, Y 36.3200, Z -7.1667, A 0.000, B 0.000, C 0.000 }
gfCNCPoint5[9271] = {X 386.9552, Y 35.0297, Z -7.1667, A 0.000, B 0.000, C 0.000 }
gfCNCPoint5[9272] = {X 386.3481, Y 33.9740, Z -7.1667, A 0.000, B 0.000, C 0.000 }
gfCNCPoint5[9273] = {X 388.4287, Y 32.7776, Z -7.1667, A 0.000, B 0.000, C 0.000 }
gfCNCPoint5[9274] = {X 384.7461, Y 26.3737, Z -7.1667, A 0.000, B 0.000, C 0.000 }
gfCNCPoint5[9275] = {X 384.6169, Y 28.7736, Z -7.1667, A 0.000, B 0.000, C 0.000 }
gfCNCPoint5[9276] = {X 384.3641, Y 31.1637, Z -7.1667, A 0.000, B 0.000, C 0.000 }
gfCNCPoint5[9277] = {X 383.9882, Y 33.5376, Z -7.1667, A 0.000, B 0.000, C 0.000 }
gfCNCPoint5[9278] = {X 383.9112, Y 33.9435, Z -7.1667, A 0.000, B 0.000, C 0.000 }
gfCNCPoint5[9279] = {X 383.8307, Y 34.3486, Z -7.1667, A 0.000, B 0.000, C 0.000 }
gfCNCPoint5[9280] = {X 383.6809, Y 35.0545, Z -7.1667, A 0.000, B 0.000, C 0.000 }
gfCNCPoint5[9281] = {X 383.5181, Y 35.7574, Z -7.1667, A 0.000, B 0.000, C 0.000 }
gfCNCPoint5[9282] = {X 383.1281, Y 37.2469, Z -7.1667, A 0.000, B 0.000, C 0.000 }
gfCNCPoint5[9283] = {X 382.6803, Y 38.7200, Z -7.1667, A 0.000, B 0.000, C 0.000 }
gfCNCPoint5[9284] = {X 388.0597, Y 38.7200, Z -7.1667, A 0.000, B 0.000, C 0.000 }
gfCNCPoint5[9285] = {X 388.4821, Y 38.7246, Z -7.1667, A 0.000, B 0.000, C 0.000 }
gfCNCPoint5[9286] = {X 388.9043, Y 38.7385, Z -7.1667, A 0.000, B 0.000, C 0.000 }
gfCNCPoint5[9287] = {X 389.1204, Y 38.2363, Z -7.1667, A 0.000, B 0.000, C 0.000 }
gfCNCPoint5[9288] = {X 389.3552, Y 37.7427, Z -7.1667, A 0.000, B 0.000, C 0.000 }
gfCNCPoint5[9289] = {X 389.3552, Y 34.3888, Z -7.1667, A 0.000, B 0.000, C 0.000 }
gfCNCPoint5[9290] = {X 388.4287, Y 32.7776, Z -7.1667, A 0.000, B 0.000, C 0.000 }
gfCNCPoint5[9291] = {X 390.5092, Y 31.5812, Z -7.1667, A 0.000, B 0.000, C 0.000 }
gfCNCPoint5[9292] = {X 386.7085, Y 24.9718, Z -7.1667, A 0.000, B 0.000, C 0.000 }
gfCNCPoint5[9293] = {X 386.1112, Y 23.9515, Z -7.1667, A 0.000, B 0.000, C 0.000 }
gfCNCPoint5[9294] = {X 385.4981, Y 22.9408, Z -7.1667, A 0.000, B 0.000, C 0.000 }
gfCNCPoint5[9295] = {X 384.4701, Y 22.1516, Z -7.1667, A 0.000, B 0.000, C 0.000 }
gfCNCPoint5[9296] = {X 383.5327, Y 21.2569, Z -7.1667, A 0.000, B 0.000, C 0.000 }
gfCNCPoint5[9297] = {X 382.6964, Y 20.2669, Z -7.1667, A 0.000, B 0.000, C 0.000 }
gfCNCPoint5[9298] = {X 381.9711, Y 19.1930, Z -7.1667, A 0.000, B 0.000, C 0.000 }
gfCNCPoint5[9299] = {X 382.2241, Y 21.5563, Z -7.1667, A 0.000, B 0.000, C 0.000 }
gfCNCPoint5[9300] = {X 382.3495, Y 23.9298, Z -7.1667, A 0.000, B 0.000, C 0.000 }
gfCNCPoint5[9301] = {X 382.3471, Y 26.3066, Z -7.1667, A 0.000, B 0.000, C 0.000 }
gfCNCPoint5[9302] = {X 382.2030, Y 28.8433, Z -7.1667, A 0.000, B 0.000, C 0.000 }
gfCNCPoint5[9303] = {X 381.9132, Y 31.3676, Z -7.1667, A 0.000, B 0.000, C 0.000 }
gfCNCPoint5[9304] = {X 381.4787, Y 33.8710, Z -7.1667, A 0.000, B 0.000, C 0.000 }
gfCNCPoint5[9305] = {X 380.9972, Y 35.9397, Z -7.1667, A 0.000, B 0.000, C 0.000 }
gfCNCPoint5[9306] = {X 380.3981, Y 37.9774, Z -7.1667, A 0.000, B 0.000, C 0.000 }
gfCNCPoint5[9307] = {X 379.8425, Y 39.5621, Z -7.1667, A 0.000, B 0.000, C 0.000 }
gfCNCPoint5[9308] = {X 379.2157, Y 41.1200, Z -7.1667, A 0.000, B 0.000, C 0.000 }
gfCNCPoint5[9309] = {X 388.0597, Y 41.1200, Z -7.1667, A 0.000, B 0.000, C 0.000 }
gfCNCPoint5[9310] = {X 389.3256, Y 41.1675, Z -7.1667, A 0.000, B 0.000, C 0.000 }
gfCNCPoint5[9311] = {X 390.5843, Y 41.3099, Z -7.1667, A 0.000, B 0.000, C 0.000 }
gfCNCPoint5[9312] = {X 391.0709, Y 39.7838, Z -7.1667, A 0.000, B 0.000, C 0.000 }
gfCNCPoint5[9313] = {X 391.7552, Y 38.3355, Z -7.1667, A 0.000, B 0.000, C 0.000 }
gfCNCPoint5[9314] = {X 391.7552, Y 33.7480, Z -7.1667, A 0.000, B 0.000, C 0.000 }
gfCNCPoint5[9315] = {X 390.5092, Y 31.5812, Z -7.1667, A 0.000, B 0.000, C 0.000 }
gfCNCPoint5[9316] = {X 392.5897, Y 30.3848, Z -7.1667, A 0.000, B 0.000, C 0.000 }
gfCNCPoint5[9317] = {X 388.7890, Y 23.7753, Z -7.1667, A 0.000, B 0.000, C 0.000 }
gfCNCPoint5[9318] = {X 388.0340, Y 22.4909, Z -7.1667, A 0.000, B 0.000, C 0.000 }
gfCNCPoint5[9319] = {X 387.2548, Y 21.2211, Z -7.1667, A 0.000, B 0.000, C 0.000 }
gfCNCPoint5[9320] = {X 386.3073, Y 20.5565, Z -7.1667, A 0.000, B 0.000, C 0.000 }
gfCNCPoint5[9321] = {X 385.4458, Y 19.7836, Z -7.1667, A 0.000, B 0.000, C 0.000 }
gfCNCPoint5[9322] = {X 384.6828, Y 18.9133, Z -7.1667, A 0.000, B 0.000, C 0.000 }
gfCNCPoint5[9323] = {X 384.0291, Y 17.9583, Z -7.1667, A 0.000, B 0.000, C 0.000 }
gfCNCPoint5[9324] = {X 383.4404, Y 16.8101, Z -7.1667, A 0.000, B 0.000, C 0.000 }
gfCNCPoint5[9325] = {X 383.0097, Y 15.5938, Z -7.1667, A 0.000, B 0.000, C 0.000 }
gfCNCPoint5[9326] = {X 382.7446, Y 14.3311, Z -7.1667, A 0.000, B 0.000, C 0.000 }
gfCNCPoint5[9327] = {X 382.6498, Y 13.0443, Z -7.1667, A 0.000, B 0.000, C 0.000 }
gfCNCPoint5[9328] = {X 382.6496, Y 12.1868, Z -7.1667, A 0.000, B 0.000, C 0.000 }
gfCNCPoint5[9329] = {X 382.6507, Y 12.0458, Z -7.1667, A 0.000, B 0.000, C 0.000 }
gfCNCPoint5[9330] = {X 382.6537, Y 11.9049, Z -7.1667, A 0.000, B 0.000, C 0.000 }
gfCNCPoint5[9331] = {X 377.7917, Y 11.9049, Z -7.1667, A 0.000, B 0.000, C 0.000 }
gfCNCPoint5[9332] = {X 378.2875, Y 13.4093, Z -7.1667, A 0.000, B 0.000, C 0.000 }
gfCNCPoint5[9333] = {X 378.7147, Y 14.9347, Z -7.1667, A 0.000, B 0.000, C 0.000 }
gfCNCPoint5[9334] = {X 379.2175, Y 17.2114, Z -7.1667, A 0.000, B 0.000, C 0.000 }
gfCNCPoint5[9335] = {X 379.5924, Y 19.5127, Z -7.1667, A 0.000, B 0.000, C 0.000 }
gfCNCPoint5[9336] = {X 379.8714, Y 22.2888, Z -7.1667, A 0.000, B 0.000, C 0.000 }
gfCNCPoint5[9337] = {X 379.9643, Y 25.0774, Z -7.1667, A 0.000, B 0.000, C 0.000 }
gfCNCPoint5[9338] = {X 379.8707, Y 27.8660, Z -7.1667, A 0.000, B 0.000, C 0.000 }
gfCNCPoint5[9339] = {X 379.5911, Y 30.6422, Z -7.1667, A 0.000, B 0.000, C 0.000 }
gfCNCPoint5[9340] = {X 379.1267, Y 33.3934, Z -7.1667, A 0.000, B 0.000, C 0.000 }
gfCNCPoint5[9341] = {X 378.5763, Y 35.7001, Z -7.1667, A 0.000, B 0.000, C 0.000 }
gfCNCPoint5[9342] = {X 377.8697, Y 37.9639, Z -7.1667, A 0.000, B 0.000, C 0.000 }
gfCNCPoint5[9343] = {X 377.0100, Y 40.1741, Z -7.1667, A 0.000, B 0.000, C 0.000 }
gfCNCPoint5[9344] = {X 376.2284, Y 41.8693, Z -7.1667, A 0.000, B 0.000, C 0.000 }
gfCNCPoint5[9345] = {X 375.3567, Y 43.5200, Z -7.1667, A 0.000, B 0.000, C 0.000 }
gfCNCPoint5[9346] = {X 388.0597, Y 43.5200, Z -7.1667, A 0.000, B 0.000, C 0.000 }
gfCNCPoint5[9347] = {X 389.6072, Y 43.6029, Z -7.1667, A 0.000, B 0.000, C 0.000 }
gfCNCPoint5[9348] = {X 391.1370, Y 43.8508, Z -7.1667, A 0.000, B 0.000, C 0.000 }
gfCNCPoint5[9349] = {X 392.6316, Y 44.2607, Z -7.1667, A 0.000, B 0.000, C 0.000 }
gfCNCPoint5[9350] = {X 392.7236, Y 42.8756, Z -7.1667, A 0.000, B 0.000, C 0.000 }
gfCNCPoint5[9351] = {X 393.0129, Y 41.5179, Z -7.1667, A 0.000, B 0.000, C 0.000 }
gfCNCPoint5[9352] = {X 393.4934, Y 40.2155, Z -7.1667, A 0.000, B 0.000, C 0.000 }
gfCNCPoint5[9353] = {X 394.1552, Y 38.9952, Z -7.1667, A 0.000, B 0.000, C 0.000 }
gfCNCPoint5[9354] = {X 394.1552, Y 33.1071, Z -7.1667, A 0.000, B 0.000, C 0.000 }
gfCNCPoint5[9355] = {X 392.5897, Y 30.3848, Z -7.1667, A 0.000, B 0.000, C 0.000 }
gfCNCPoint5[9356] = {X 394.6703, Y 29.1884, Z -7.1667, A 0.000, B 0.000, C 0.000 }
gfCNCPoint5[9357] = {X 390.8695, Y 22.5789, Z -7.1667, A 0.000, B 0.000, C 0.000 }
gfCNCPoint5[9358] = {X 390.0503, Y 21.1867, Z -7.1667, A 0.000, B 0.000, C 0.000 }
gfCNCPoint5[9359] = {X 389.2033, Y 19.8111, Z -7.1667, A 0.000, B 0.000, C 0.000 }
gfCNCPoint5[9360] = {X 389.0602, Y 19.6007, Z -7.1667, A 0.000, B 0.000, C 0.000 }
gfCNCPoint5[9361] = {X 388.9027, Y 19.4010, Z -7.1667, A 0.000, B 0.000, C 0.000 }
gfCNCPoint5[9362] = {X 387.8149, Y 18.6890, Z -7.1667, A 0.000, B 0.000, C 0.000 }
gfCNCPoint5[9363] = {X 386.8711, Y 17.7950, Z -7.1667, A 0.000, B 0.000, C 0.000 }
gfCNCPoint5[9364] = {X 386.1014, Y 16.7473, Z -7.1667, A 0.000, B 0.000, C 0.000 }
gfCNCPoint5[9365] = {X 385.5303, Y 15.5794, Z -7.1667, A 0.000, B 0.000, C 0.000 }
gfCNCPoint5[9366] = {X 385.1760, Y 14.3286, Z -7.1667, A 0.000, B 0.000, C 0.000 }
gfCNCPoint5[9367] = {X 385.0498, Y 13.0347, Z -7.1667, A 0.000, B 0.000, C 0.000 }
gfCNCPoint5[9368] = {X 385.0496, Y 12.1868, Z -7.1667, A 0.000, B 0.000, C 0.000 }
gfCNCPoint5[9369] = {X 385.0504, Y 12.0808, Z -7.1667, A 0.000, B 0.000, C 0.000 }
gfCNCPoint5[9370] = {X 385.0527, Y 11.9748, Z -7.1667, A 0.000, B 0.000, C 0.000 }
gfCNCPoint5[9371] = {X 385.1994, Y 10.7176, Z -7.1667, A 0.000, B 0.000, C 0.000 }
gfCNCPoint5[9372] = {X 385.5617, Y 9.5049, Z -7.1667, A 0.000, B 0.000, C 0.000 }
gfCNCPoint5[9373] = {X 374.1977, Y 9.5049, Z -7.1667, A 0.000, B 0.000, C 0.000 }
gfCNCPoint5[9374] = {X 374.9064, Y 11.0884, Z -7.1667, A 0.000, B 0.000, C 0.000 }
gfCNCPoint5[9375] = {X 375.5298, Y 12.7074, Z -7.1667, A 0.000, B 0.000, C 0.000 }
gfCNCPoint5[9376] = {X 375.9908, Y 14.1058, Z -7.1667, A 0.000, B 0.000, C 0.000 }
gfCNCPoint5[9377] = {X 376.3881, Y 15.5236, Z -7.1667, A 0.000, B 0.000, C 0.000 }
gfCNCPoint5[9378] = {X 376.9916, Y 18.3835, Z -7.1667, A 0.000, B 0.000, C 0.000 }
gfCNCPoint5[9379] = {X 377.3811, Y 21.2803, Z -7.1667, A 0.000, B 0.000, C 0.000 }
gfCNCPoint5[9380] = {X 377.5546, Y 24.1980, Z -7.1667, A 0.000, B 0.000, C 0.000 }
gfCNCPoint5[9381] = {X 377.5110, Y 27.1206, Z -7.1667, A 0.000, B 0.000, C 0.000 }
gfCNCPoint5[9382] = {X 377.2505, Y 30.0318, Z -7.1667, A 0.000, B 0.000, C 0.000 }
gfCNCPoint5[9383] = {X 376.7747, Y 32.9157, Z -7.1667, A 0.000, B 0.000, C 0.000 }
gfCNCPoint5[9384] = {X 376.1769, Y 35.3683, Z -7.1667, A 0.000, B 0.000, C 0.000 }
gfCNCPoint5[9385] = {X 375.3893, Y 37.7667, Z -7.1667, A 0.000, B 0.000, C 0.000 }
gfCNCPoint5[9386] = {X 374.4168, Y 40.0962, Z -7.1667, A 0.000, B 0.000, C 0.000 }
gfCNCPoint5[9387] = {X 373.2653, Y 42.3426, Z -7.1667, A 0.000, B 0.000, C 0.000 }
gfCNCPoint5[9388] = {X 372.1896, Y 44.1175, Z -7.1667, A 0.000, B 0.000, C 0.000 }
gfCNCPoint5[9389] = {X 371.0020, Y 45.8196, Z -7.1667, A 0.000, B 0.000, C 0.000 }
gfCNCPoint5[9390] = {X 370.9161, Y 45.9351, Z -7.1667, A 0.000, B 0.000, C 0.000 }
gfCNCPoint5[9391] = {X 371.2176, Y 45.9238, Z -7.1667, A 0.000, B 0.000, C 0.000 }
gfCNCPoint5[9392] = {X 371.5193, Y 45.9200, Z -7.1667, A 0.000, B 0.000, C 0.000 }
gfCNCPoint5[9393] = {X 388.0597, Y 45.9200, Z -7.1667, A 0.000, B 0.000, C 0.000 }
gfCNCPoint5[9394] = {X 389.4143, Y 45.9962, Z -7.1667, A 0.000, B 0.000, C 0.000 }
gfCNCPoint5[9395] = {X 390.7519, Y 46.2238, Z -7.1667, A 0.000, B 0.000, C 0.000 }
gfCNCPoint5[9396] = {X 392.0555, Y 46.6000, Z -7.1667, A 0.000, B 0.000, C 0.000 }
gfCNCPoint5[9397] = {X 393.3087, Y 47.1200, Z -7.1667, A 0.000, B 0.000, C 0.000 }
gfCNCPoint5[9398] = {X 394.2237, Y 46.7243, Z -7.1667, A 0.000, B 0.000, C 0.000 }
gfCNCPoint5[9399] = {X 395.1681, Y 46.4053, Z -7.1667, A 0.000, B 0.000, C 0.000 }
gfCNCPoint5[9400] = {X 395.0678, Y 45.7292, Z -7.1667, A 0.000, B 0.000, C 0.000 }
gfCNCPoint5[9401] = {X 395.0314, Y 45.0468, Z -7.1667, A 0.000, B 0.000, C 0.000 }
gfCNCPoint5[9402] = {X 395.0316, Y 44.1297, Z -7.1667, A 0.000, B 0.000, C 0.000 }
gfCNCPoint5[9403] = {X 395.1397, Y 42.9565, Z -7.1667, A 0.000, B 0.000, C 0.000 }
gfCNCPoint5[9404] = {X 395.4356, Y 41.8161, Z -7.1667, A 0.000, B 0.000, C 0.000 }
gfCNCPoint5[9405] = {X 395.9116, Y 40.7384, Z -7.1667, A 0.000, B 0.000, C 0.000 }
gfCNCPoint5[9406] = {X 396.5552, Y 39.7516, Z -7.1667, A 0.000, B 0.000, C 0.000 }
gfCNCPoint5[9407] = {X 396.5552, Y 32.4663, Z -7.1667, A 0.000, B 0.000, C 0.000 }
gfCNCPoint5[9408] = {X 394.6703, Y 29.1884, Z -7.1667, A 0.000, B 0.000, C 0.000 }
gfCNCPoint5[9409] = {X 396.7508, Y 27.9920, Z -7.1667, A 0.000, B 0.000, C 0.000 }
gfCNCPoint5[9410] = {X 392.9501, Y 21.3825, Z -7.1667, A 0.000, B 0.000, C 0.000 }
gfCNCPoint5[9411] = {X 392.1064, Y 19.9489, Z -7.1667, A 0.000, B 0.000, C 0.000 }
gfCNCPoint5[9412] = {X 391.2343, Y 18.5324, Z -7.1667, A 0.000, B 0.000, C 0.000 }
gfCNCPoint5[9413] = {X 390.8251, Y 17.9599, Z -7.1667, A 0.000, B 0.000, C 0.000 }
gfCNCPoint5[9414] = {X 390.3518, Y 17.4392, Z -7.1667, A 0.000, B 0.000, C 0.000 }
gfCNCPoint5[9415] = {X 389.5420, Y 16.9835, Z -7.1667, A 0.000, B 0.000, C 0.000 }
gfCNCPoint5[9416] = {X 388.8333, Y 16.3825, Z -7.1667, A 0.000, B 0.000, C 0.000 }
gfCNCPoint5[9417] = {X 388.2514, Y 15.6580, Z -7.1667, A 0.000, B 0.000, C 0.000 }
gfCNCPoint5[9418] = {X 387.8173, Y 14.8364, Z -7.1667, A 0.000, B 0.000, C 0.000 }
gfCNCPoint5[9419] = {X 387.5469, Y 13.9474, Z -7.1667, A 0.000, B 0.000, C 0.000 }
gfCNCPoint5[9420] = {X 387.4498, Y 13.0232, Z -7.1667, A 0.000, B 0.000, C 0.000 }
gfCNCPoint5[9421] = {X 387.4496, Y 12.1868, Z -7.1667, A 0.000, B 0.000, C 0.000 }
gfCNCPoint5[9422] = {X 387.5362, Y 11.2717, Z -7.1667, A 0.000, B 0.000, C 0.000 }
gfCNCPoint5[9423] = {X 387.7929, Y 10.3890, Z -7.1667, A 0.000, B 0.000, C 0.000 }
gfCNCPoint5[9424] = {X 388.2376, Y 9.5280, Z -7.1667, A 0.000, B 0.000, C 0.000 }
gfCNCPoint5[9425] = {X 388.8437, Y 8.7718, Z -7.1667, A 0.000, B 0.000, C 0.000 }
gfCNCPoint5[9426] = {X 389.5873, Y 8.1503, Z -7.1667, A 0.000, B 0.000, C 0.000 }
gfCNCPoint5[9427] = {X 390.4390, Y 7.6879, Z -7.1667, A 0.000, B 0.000, C 0.000 }
gfCNCPoint5[9428] = {X 391.3653, Y 7.4030, Z -7.1667, A 0.000, B 0.000, C 0.000 }
gfCNCPoint5[9429] = {X 392.3296, Y 7.3068, Z -7.1667, A 0.000, B 0.000, C 0.000 }
gfCNCPoint5[9430] = {X 399.1118, Y 7.3068, Z -7.1667, A 0.000, B 0.000, C 0.000 }
gfCNCPoint5[9431] = {X 400.0638, Y 7.4006, Z -7.1667, A 0.000, B 0.000, C 0.000 }
gfCNCPoint5[9432] = {X 400.9793, Y 7.6783, Z -7.1667, A 0.000, B 0.000, C 0.000 }
gfCNCPoint5[9433] = {X 401.8229, Y 8.1292, Z -7.1667, A 0.000, B 0.000, C 0.000 }
gfCNCPoint5[9434] = {X 402.5624, Y 8.7361, Z -7.1667, A 0.000, B 0.000, C 0.000 }
gfCNCPoint5[9435] = {X 403.1693, Y 9.4756, Z -7.1667, A 0.000, B 0.000, C 0.000 }
gfCNCPoint5[9436] = {X 403.6203, Y 10.3193, Z -7.1667, A 0.000, B 0.000, C 0.000 }
gfCNCPoint5[9437] = {X 403.8980, Y 11.2348, Z -7.1667, A 0.000, B 0.000, C 0.000 }
gfCNCPoint5[9438] = {X 403.9918, Y 12.1868, Z -7.1667, A 0.000, B 0.000, C 0.000 }
gfCNCPoint5[9439] = {X 403.9915, Y 13.0237, Z -7.1667, A 0.000, B 0.000, C 0.000 }
gfCNCPoint5[9440] = {X 403.9016, Y 13.9115, Z -7.1667, A 0.000, B 0.000, C 0.000 }
gfCNCPoint5[9441] = {X 403.6516, Y 14.7680, Z -7.1667, A 0.000, B 0.000, C 0.000 }
gfCNCPoint5[9442] = {X 405.3642, Y 17.7418, Z -7.1667, A 0.000, B 0.000, C 0.000 }
gfCNCPoint5[9443] = {X 407.2442, Y 14.6968, Z -7.1667, A 0.000, B 0.000, C 0.000 }
gfCNCPoint5[9444] = {X 407.0141, Y 13.8721, Z -7.1667, A 0.000, B 0.000, C 0.000 }
gfCNCPoint5[9445] = {X 406.9317, Y 13.0199, Z -7.1667, A 0.000, B 0.000, C 0.000 }
gfCNCPoint5[9446] = {X 406.9315, Y 12.1868, Z -7.1667, A 0.000, B 0.000, C 0.000 }
gfCNCPoint5[9447] = {X 407.0253, Y 11.2348, Z -7.1667, A 0.000, B 0.000, C 0.000 }
gfCNCPoint5[9448] = {X 407.3030, Y 10.3193, Z -7.1667, A 0.000, B 0.000, C 0.000 }
gfCNCPoint5[9449] = {X 407.7540, Y 9.4756, Z -7.1667, A 0.000, B 0.000, C 0.000 }
gfCNCPoint5[9450] = {X 408.3609, Y 8.7361, Z -7.1667, A 0.000, B 0.000, C 0.000 }
gfCNCPoint5[9451] = {X 409.1004, Y 8.1292, Z -7.1667, A 0.000, B 0.000, C 0.000 }
gfCNCPoint5[9452] = {X 409.9440, Y 7.6783, Z -7.1667, A 0.000, B 0.000, C 0.000 }
gfCNCPoint5[9453] = {X 410.8595, Y 7.4006, Z -7.1667, A 0.000, B 0.000, C 0.000 }
gfCNCPoint5[9454] = {X 411.8115, Y 7.3068, Z -7.1667, A 0.000, B 0.000, C 0.000 }
gfCNCPoint5[9455] = {X 419.3245, Y 7.3068, Z -7.1667, A 0.000, B 0.000, C 0.000 }
gfCNCPoint5[9456] = {X 420.2888, Y 7.4030, Z -7.1667, A 0.000, B 0.000, C 0.000 }
gfCNCPoint5[9457] = {X 421.2151, Y 7.6879, Z -7.1667, A 0.000, B 0.000, C 0.000 }
gfCNCPoint5[9458] = {X 422.0668, Y 8.1503, Z -7.1667, A 0.000, B 0.000, C 0.000 }
gfCNCPoint5[9459] = {X 422.8104, Y 8.7718, Z -7.1667, A 0.000, B 0.000, C 0.000 }
gfCNCPoint5[9460] = {X 423.4165, Y 9.5280, Z -7.1667, A 0.000, B 0.000, C 0.000 }
gfCNCPoint5[9461] = {X 423.8612, Y 10.3890, Z -7.1667, A 0.000, B 0.000, C 0.000 }
gfCNCPoint5[9462] = {X 424.1179, Y 11.2717, Z -7.1667, A 0.000, B 0.000, C 0.000 }
gfCNCPoint5[9463] = {X 424.2045, Y 12.1868, Z -7.1667, A 0.000, B 0.000, C 0.000 }
gfCNCPoint5[9464] = {X 424.2045, Y 12.9780, Z -7.1667, A 0.000, B 0.000, C 0.000 }
gfCNCPoint5[9465] = {X 424.1064, Y 13.9308, Z -7.1667, A 0.000, B 0.000, C 0.000 }
gfCNCPoint5[9466] = {X 423.8263, Y 14.8468, Z -7.1667, A 0.000, B 0.000, C 0.000 }
gfCNCPoint5[9467] = {X 423.3748, Y 15.6916, Z -7.1667, A 0.000, B 0.000, C 0.000 }
gfCNCPoint5[9468] = {X 422.7687, Y 16.4333, Z -7.1667, A 0.000, B 0.000, C 0.000 }
gfCNCPoint5[9469] = {X 422.0309, Y 17.0442, Z -7.1667, A 0.000, B 0.000, C 0.000 }
gfCNCPoint5[9470] = {X 421.1891, Y 17.5012, Z -7.1667, A 0.000, B 0.000, C 0.000 }
gfCNCPoint5[9471] = {X 420.5411, Y 18.3845, Z -7.1667, A 0.000, B 0.000, C 0.000 }
gfCNCPoint5[9472] = {X 419.9522, Y 19.3082, Z -7.1667, A 0.000, B 0.000, C 0.000 }
gfCNCPoint5[9473] = {X 414.1625, Y 28.6207, Z -7.1667, A 0.000, B 0.000, C 0.000 }
gfCNCPoint5[9474] = {X 422.3153, Y 33.6894, Z -7.1667, A 0.000, B 0.000, C 0.000 }
gfCNCPoint5[9475] = {X 421.8957, Y 34.3643, Z -7.1667, A 0.000, B 0.000, C 0.000 }
gfCNCPoint5[9476] = {X 422.1481, Y 34.0989, Z -7.1667, A 0.000, B 0.000, C 0.000 }
gfCNCPoint5[9477] = {X 422.4071, Y 33.8400, Z -7.1667, A 0.000, B 0.000, C 0.000 }
gfCNCPoint5[9478] = {X 422.3611, Y 33.7648, Z -7.1667, A 0.000, B 0.000, C 0.000 }
gfCNCPoint5[9479] = {X 422.3153, Y 33.6894, Z -7.1667, A 0.000, B 0.000, C 0.000 }
gfCNCPoint5[9480] = {X 420.2771, Y 32.4222, Z -7.1667, A 0.000, B 0.000, C 0.000 }
gfCNCPoint5[9481] = {X 419.3081, Y 33.9809, Z -7.1667, A 0.000, B 0.000, C 0.000 }
gfCNCPoint5[9482] = {X 419.3083, Y 38.3384, Z -7.1667, A 0.000, B 0.000, C 0.000 }
gfCNCPoint5[9483] = {X 419.9587, Y 39.7074, Z -7.1667, A 0.000, B 0.000, C 0.000 }
gfCNCPoint5[9484] = {X 420.4342, Y 41.1465, Z -7.1667, A 0.000, B 0.000, C 0.000 }
gfCNCPoint5[9485] = {X 420.6283, Y 41.1585, Z -7.1667, A 0.000, B 0.000, C 0.000 }
gfCNCPoint5[9486] = {X 420.8222, Y 41.1728, Z -7.1667, A 0.000, B 0.000, C 0.000 }
gfCNCPoint5[9487] = {X 421.2847, Y 39.7569, Z -7.1667, A 0.000, B 0.000, C 0.000 }
gfCNCPoint5[9488] = {X 421.9179, Y 38.4087, Z -7.1667, A 0.000, B 0.000, C 0.000 }
gfCNCPoint5[9489] = {X 422.7123, Y 37.1487, Z -7.1667, A 0.000, B 0.000, C 0.000 }
gfCNCPoint5[9490] = {X 423.6557, Y 35.9960, Z -7.1667, A 0.000, B 0.000, C 0.000 }
gfCNCPoint5[9491] = {X 424.3430, Y 35.3119, Z -7.1667, A 0.000, B 0.000, C 0.000 }
gfCNCPoint5[9492] = {X 425.0829, Y 34.6852, Z -7.1667, A 0.000, B 0.000, C 0.000 }
gfCNCPoint5[9493] = {X 425.4251, Y 34.0154, Z -7.1667, A 0.000, B 0.000, C 0.000 }
gfCNCPoint5[9494] = {X 424.8780, Y 33.2451, Z -7.1667, A 0.000, B 0.000, C 0.000 }
gfCNCPoint5[9495] = {X 424.3698, Y 32.4488, Z -7.1667, A 0.000, B 0.000, C 0.000 }
gfCNCPoint5[9496] = {X 423.3889, Y 30.6028, Z -7.1667, A 0.000, B 0.000, C 0.000 }
gfCNCPoint5[9497] = {X 422.6158, Y 28.6606, Z -7.1667, A 0.000, B 0.000, C 0.000 }
gfCNCPoint5[9498] = {X 420.2771, Y 32.4222, Z -7.1667, A 0.000, B 0.000, C 0.000 }
gfCNCPoint5[9499] = {X 418.2389, Y 31.1550, Z -7.1667, A 0.000, B 0.000, C 0.000 }
gfCNCPoint5[9500] = {X 416.9080, Y 33.2958, Z -7.1667, A 0.000, B 0.000, C 0.000 }
gfCNCPoint5[9501] = {X 416.9084, Y 38.9950, Z -7.1667, A 0.000, B 0.000, C 0.000 }
gfCNCPoint5[9502] = {X 417.4897, Y 40.0483, Z -7.1667, A 0.000, B 0.000, C 0.000 }
gfCNCPoint5[9503] = {X 417.9375, Y 41.1649, Z -7.1667, A 0.000, B 0.000, C 0.000 }
gfCNCPoint5[9504] = {X 418.2451, Y 42.3280, Z -7.1667, A 0.000, B 0.000, C 0.000 }
gfCNCPoint5[9505] = {X 418.4078, Y 43.5200, Z -7.1667, A 0.000, B 0.000, C 0.000 }
gfCNCPoint5[9506] = {X 419.4886, Y 43.5200, Z -7.1667, A 0.000, B 0.000, C 0.000 }
gfCNCPoint5[9507] = {X 421.1752, Y 43.6186, Z -7.1667, A 0.000, B 0.000, C 0.000 }
gfCNCPoint5[9508] = {X 422.8389, Y 43.9129, Z -7.1667, A 0.000, B 0.000, C 0.000 }
gfCNCPoint5[9509] = {X 423.0005, Y 42.4234, Z -7.1667, A 0.000, B 0.000, C 0.000 }
gfCNCPoint5[9510] = {X 423.3900, Y 40.9766, Z -7.1667, A 0.000, B 0.000, C 0.000 }
gfCNCPoint5[9511] = {X 423.9980, Y 39.6073, Z -7.1667, A 0.000, B 0.000, C 0.000 }
gfCNCPoint5[9512] = {X 424.8102, Y 38.3482, Z -7.1667, A 0.000, B 0.000, C 0.000 }
gfCNCPoint5[9513] = {X 425.8068, Y 37.2295, Z -7.1667, A 0.000, B 0.000, C 0.000 }
gfCNCPoint5[9514] = {X 426.9642, Y 36.2780, Z -7.1667, A 0.000, B 0.000, C 0.000 }
gfCNCPoint5[9515] = {X 428.2754, Y 33.7114, Z -7.1667, A 0.000, B 0.000, C 0.000 }
gfCNCPoint5[9516] = {X 427.2117, Y 32.3944, Z -7.1667, A 0.000, B 0.000, C 0.000 }
gfCNCPoint5[9517] = {X 426.2869, Y 30.9764, Z -7.1667, A 0.000, B 0.000, C 0.000 }
gfCNCPoint5[9518] = {X 425.5106, Y 29.4719, Z -7.1667, A 0.000, B 0.000, C 0.000 }
gfCNCPoint5[9519] = {X 424.8909, Y 27.8965, Z -7.1667, A 0.000, B 0.000, C 0.000 }
gfCNCPoint5[9520] = {X 424.8186, Y 27.6762, Z -7.1667, A 0.000, B 0.000, C 0.000 }
gfCNCPoint5[9521] = {X 424.7494, Y 27.4549, Z -7.1667, A 0.000, B 0.000, C 0.000 }
gfCNCPoint5[9522] = {X 424.3067, Y 25.6994, Z -7.1667, A 0.000, B 0.000, C 0.000 }
gfCNCPoint5[9523] = {X 424.0106, Y 23.9133, Z -7.1667, A 0.000, B 0.000, C 0.000 }
gfCNCPoint5[9524] = {X 423.8630, Y 22.1089, Z -7.1667, A 0.000, B 0.000, C 0.000 }
gfCNCPoint5[9525] = {X 418.2389, Y 31.1550, Z -7.1667, A 0.000, B 0.000, C 0.000 }
gfCNCPoint5[9526] = {X 416.2007, Y 29.8879, Z -7.1667, A 0.000, B 0.000, C 0.000 }
gfCNCPoint5[9527] = {X 414.5080, Y 32.6106, Z -7.1667, A 0.000, B 0.000, C 0.000 }
gfCNCPoint5[9528] = {X 414.5084, Y 39.7464, Z -7.1667, A 0.000, B 0.000, C 0.000 }
gfCNCPoint5[9529] = {X 415.1571, Y 40.7517, Z -7.1667, A 0.000, B 0.000, C 0.000 }
gfCNCPoint5[9530] = {X 415.6352, Y 41.8484, Z -7.1667, A 0.000, B 0.000, C 0.000 }
gfCNCPoint5[9531] = {X 415.9303, Y 43.0078, Z -7.1667, A 0.000, B 0.000, C 0.000 }
gfCNCPoint5[9532] = {X 416.0347, Y 44.1997, Z -7.1667, A 0.000, B 0.000, C 0.000 }
gfCNCPoint5[9533] = {X 416.0347, Y 45.0000, Z -7.1667, A 0.000, B 0.000, C 0.000 }
gfCNCPoint5[9534] = {X 416.0201, Y 45.4609, Z -7.1667, A 0.000, B 0.000, C 0.000 }
gfCNCPoint5[9535] = {X 415.9763, Y 45.9200, Z -7.1667, A 0.000, B 0.000, C 0.000 }
gfCNCPoint5[9536] = {X 419.4886, Y 45.9200, Z -7.1667, A 0.000, B 0.000, C 0.000 }
gfCNCPoint5[9537] = {X 420.8957, Y 46.0022, Z -7.1667, A 0.000, B 0.000, C 0.000 }
gfCNCPoint5[9538] = {X 422.2836, Y 46.2478, Z -7.1667, A 0.000, B 0.000, C 0.000 }
gfCNCPoint5[9539] = {X 423.4822, Y 46.5992, Z -7.1667, A 0.000, B 0.000, C 0.000 }
gfCNCPoint5[9540] = {X 424.6380, Y 47.0725, Z -7.1667, A 0.000, B 0.000, C 0.000 }
gfCNCPoint5[9541] = {X 425.7388, Y 47.6626, Z -7.1667, A 0.000, B 0.000, C 0.000 }
gfCNCPoint5[9542] = {X 425.4600, Y 46.7984, Z -7.1667, A 0.000, B 0.000, C 0.000 }
gfCNCPoint5[9543] = {X 425.2910, Y 45.9063, Z -7.1667, A 0.000, B 0.000, C 0.000 }
gfCNCPoint5[9544] = {X 425.2344, Y 45.0000, Z -7.1667, A 0.000, B 0.000, C 0.000 }
gfCNCPoint5[9545] = {X 425.2344, Y 44.2089, Z -7.1667, A 0.000, B 0.000, C 0.000 }
gfCNCPoint5[9546] = {X 425.2353, Y 44.0976, Z -7.1667, A 0.000, B 0.000, C 0.000 }
gfCNCPoint5[9547] = {X 425.2378, Y 43.9863, Z -7.1667, A 0.000, B 0.000, C 0.000 }
gfCNCPoint5[9548] = {X 425.3770, Y 42.7748, Z -7.1667, A 0.000, B 0.000, C 0.000 }
gfCNCPoint5[9549] = {X 425.7165, Y 41.6036, Z -7.1667, A 0.000, B 0.000, C 0.000 }
gfCNCPoint5[9550] = {X 426.2468, Y 40.5054, Z -7.1667, A 0.000, B 0.000, C 0.000 }
gfCNCPoint5[9551] = {X 426.9528, Y 39.5112, Z -7.1667, A 0.000, B 0.000, C 0.000 }
gfCNCPoint5[9552] = {X 427.8150, Y 38.6488, Z -7.1667, A 0.000, B 0.000, C 0.000 }
gfCNCPoint5[9553] = {X 428.8090, Y 37.9424, Z -7.1667, A 0.000, B 0.000, C 0.000 }
gfCNCPoint5[9554] = {X 431.2061, Y 33.2502, Z -7.1667, A 0.000, B 0.000, C 0.000 }
gfCNCPoint5[9555] = {X 430.0997, Y 32.1509, Z -7.1667, A 0.000, B 0.000, C 0.000 }
gfCNCPoint5[9556] = {X 429.1198, Y 30.9375, Z -7.1667, A 0.000, B 0.000, C 0.000 }
gfCNCPoint5[9557] = {X 428.2781, Y 29.6245, Z -7.1667, A 0.000, B 0.000, C 0.000 }
gfCNCPoint5[9558] = {X 427.5846, Y 28.2275, Z -7.1667, A 0.000, B 0.000, C 0.000 }
gfCNCPoint5[9559] = {X 427.0476, Y 26.7632, Z -7.1667, A 0.000, B 0.000, C 0.000 }
gfCNCPoint5[9560] = {X 426.6549, Y 25.2030, Z -7.1667, A 0.000, B 0.000, C 0.000 }
gfCNCPoint5[9561] = {X 426.3921, Y 23.6158, Z -7.1667, A 0.000, B 0.000, C 0.000 }
gfCNCPoint5[9562] = {X 426.2611, Y 22.0122, Z -7.1667, A 0.000, B 0.000, C 0.000 }
gfCNCPoint5[9563] = {X 426.2912, Y 19.8886, Z -7.1667, A 0.000, B 0.000, C 0.000 }
gfCNCPoint5[9564] = {X 426.5522, Y 17.7809, Z -7.1667, A 0.000, B 0.000, C 0.000 }
gfCNCPoint5[9565] = {X 427.0408, Y 15.7141, Z -7.1667, A 0.000, B 0.000, C 0.000 }
gfCNCPoint5[9566] = {X 427.6624, Y 14.0037, Z -7.1667, A 0.000, B 0.000, C 0.000 }
gfCNCPoint5[9567] = {X 428.4893, Y 12.3827, Z -7.1667, A 0.000, B 0.000, C 0.000 }
gfCNCPoint5[9568] = {X 429.5090, Y 10.8754, Z -7.1667, A 0.000, B 0.000, C 0.000 }
gfCNCPoint5[9569] = {X 430.7062, Y 9.5049, Z -7.1667, A 0.000, B 0.000, C 0.000 }
gfCNCPoint5[9570] = {X 426.0924, Y 9.5049, Z -7.1667, A 0.000, B 0.000, C 0.000 }
gfCNCPoint5[9571] = {X 426.3754, Y 10.3750, Z -7.1667, A 0.000, B 0.000, C 0.000 }
gfCNCPoint5[9572] = {X 426.5470, Y 11.2737, Z -7.1667, A 0.000, B 0.000, C 0.000 }
gfCNCPoint5[9573] = {X 426.6045, Y 12.1868, Z -7.1667, A 0.000, B 0.000, C 0.000 }
gfCNCPoint5[9574] = {X 426.6045, Y 12.9845, Z -7.1667, A 0.000, B 0.000, C 0.000 }
gfCNCPoint5[9575] = {X 426.4820, Y 14.2867, Z -7.1667, A 0.000, B 0.000, C 0.000 }
gfCNCPoint5[9576] = {X 426.1304, Y 15.5464, Z -7.1667, A 0.000, B 0.000, C 0.000 }
gfCNCPoint5[9577] = {X 425.5608, Y 16.7238, Z -7.1667, A 0.000, B 0.000, C 0.000 }
gfCNCPoint5[9578] = {X 424.7914, Y 17.7814, Z -7.1667, A 0.000, B 0.000, C 0.000 }
gfCNCPoint5[9579] = {X 423.8464, Y 18.6856, Z -7.1667, A 0.000, B 0.000, C 0.000 }
gfCNCPoint5[9580] = {X 422.7560, Y 19.4078, Z -7.1667, A 0.000, B 0.000, C 0.000 }
gfCNCPoint5[9581] = {X 422.3663, Y 19.9718, Z -7.1667, A 0.000, B 0.000, C 0.000 }
gfCNCPoint5[9582] = {X 422.0038, Y 20.5537, Z -7.1667, A 0.000, B 0.000, C 0.000 }
gfCNCPoint5[9583] = {X 416.2007, Y 29.8879, Z -7.1667, A 0.000, B 0.000, C 0.000 }
gfCNCPoint5[9584] = {X 414.1625, Y 28.6207, Z -7.1667, A 0.000, B 0.000, C 0.000 }
gfCNCPoint5[9585] = {X 412.1079, Y 31.9255, Z -7.1667, A 0.000, B 0.000, C 0.000 }
gfCNCPoint5[9586] = {X 412.1085, Y 40.6514, Z -7.1667, A 0.000, B 0.000, C 0.000 }
gfCNCPoint5[9587] = {X 412.7503, Y 41.4079, Z -7.1667, A 0.000, B 0.000, C 0.000 }
gfCNCPoint5[9588] = {X 413.2300, Y 42.2764, Z -7.1667, A 0.000, B 0.000, C 0.000 }
gfCNCPoint5[9589] = {X 413.5287, Y 43.2224, Z -7.1667, A 0.000, B 0.000, C 0.000 }
gfCNCPoint5[9590] = {X 413.6347, Y 44.2088, Z -7.1667, A 0.000, B 0.000, C 0.000 }
gfCNCPoint5[9591] = {X 413.6347, Y 45.0000, Z -7.1667, A 0.000, B 0.000, C 0.000 }
gfCNCPoint5[9592] = {X 413.6249, Y 45.3090, Z -7.1667, A 0.000, B 0.000, C 0.000 }
gfCNCPoint5[9593] = {X 413.5956, Y 45.6167, Z -7.1667, A 0.000, B 0.000, C 0.000 }
gfCNCPoint5[9594] = {X 413.3652, Y 46.5992, Z -7.1667, A 0.000, B 0.000, C 0.000 }
gfCNCPoint5[9595] = {X 412.9377, Y 47.5134, Z -7.1667, A 0.000, B 0.000, C 0.000 }
gfCNCPoint5[9596] = {X 412.3313, Y 48.3200, Z -7.1667, A 0.000, B 0.000, C 0.000 }
gfCNCPoint5[9597] = {X 411.9795, Y 47.9934, Z -7.1667, A 0.000, B 0.000, C 0.000 }
gfCNCPoint5[9598] = {X 411.3003, Y 48.5889, Z -7.1667, A 0.000, B 0.000, C 0.000 }
gfCNCPoint5[9599] = {X 410.5138, Y 49.0331, Z -7.1667, A 0.000, B 0.000, C 0.000 }
gfCNCPoint5[9600] = {X 409.6532, Y 49.3073, Z -7.1667, A 0.000, B 0.000, C 0.000 }
gfCNCPoint5[9601] = {X 408.7547, Y 49.4000, Z -7.1667, A 0.000, B 0.000, C 0.000 }
gfCNCPoint5[9602] = {X 402.3112, Y 49.4000, Z -7.1667, A 0.000, B 0.000, C 0.000 }
gfCNCPoint5[9603] = {X 401.3321, Y 49.2897, Z -7.1667, A 0.000, B 0.000, C 0.000 }
gfCNCPoint5[9604] = {X 400.4021, Y 48.9643, Z -7.1667, A 0.000, B 0.000, C 0.000 }
gfCNCPoint5[9605] = {X 399.5678, Y 48.4400, Z -7.1667, A 0.000, B 0.000, C 0.000 }
gfCNCPoint5[9606] = {X 398.8711, Y 47.7433, Z -7.1667, A 0.000, B 0.000, C 0.000 }
gfCNCPoint5[9607] = {X 398.3469, Y 46.9091, Z -7.1667, A 0.000, B 0.000, C 0.000 }
gfCNCPoint5[9608] = {X 398.0215, Y 45.9791, Z -7.1667, A 0.000, B 0.000, C 0.000 }
gfCNCPoint5[9609] = {X 397.9112, Y 45.0000, Z -7.1667, A 0.000, B 0.000, C 0.000 }
gfCNCPoint5[9610] = {X 397.9116, Y 44.1518, Z -7.1667, A 0.000, B 0.000, C 0.000 }
gfCNCPoint5[9611] = {X 398.0215, Y 43.2300, Z -7.1667, A 0.000, B 0.000, C 0.000 }
gfCNCPoint5[9612] = {X 398.3223, Y 42.3519, Z -7.1667, A 0.000, B 0.000, C 0.000 }
gfCNCPoint5[9613] = {X 398.8006, Y 41.5563, Z -7.1667, A 0.000, B 0.000, C 0.000 }
gfCNCPoint5[9614] = {X 399.4352, Y 40.8789, Z -7.1667, A 0.000, B 0.000, C 0.000 }
gfCNCPoint5[9615] = {X 399.4352, Y 31.6972, Z -7.1667, A 0.000, B 0.000, C 0.000 }
gfCNCPoint5[9616] = {X 393.3662, Y 21.1433, Z -7.1667, A 0.000, B 0.000, C 0.000 }
gfCNCPoint5[9617] = {X 392.5177, Y 19.7013, Z -7.1667, A 0.000, B 0.000, C 0.000 }
gfCNCPoint5[9618] = {X 391.6404, Y 18.2766, Z -7.1667, A 0.000, B 0.000, C 0.000 }
gfCNCPoint5[9619] = {X 391.1700, Y 17.6233, Z -7.1667, A 0.000, B 0.000, C 0.000 }
gfCNCPoint5[9620] = {X 390.6223, Y 17.0333, Z -7.1667, A 0.000, B 0.000, C 0.000 }
gfCNCPoint5[9621] = {X 389.8674, Y 16.6246, Z -7.1667, A 0.000, B 0.000, C 0.000 }
gfCNCPoint5[9622] = {X 389.2063, Y 16.0772, Z -7.1667, A 0.000, B 0.000, C 0.000 }
gfCNCPoint5[9623] = {X 388.6641, Y 15.4119, Z -7.1667, A 0.000, B 0.000, C 0.000 }
gfCNCPoint5[9624] = {X 388.2613, Y 14.6539, Z -7.1667, A 0.000, B 0.000, C 0.000 }
gfCNCPoint5[9625] = {X 388.0133, Y 13.8322, Z -7.1667, A 0.000, B 0.000, C 0.000 }
gfCNCPoint5[9626] = {X 387.9296, Y 12.9780, Z -7.1667, A 0.000, B 0.000, C 0.000 }
gfCNCPoint5[9627] = {X 387.9296, Y 12.1868, Z -7.1667, A 0.000, B 0.000, C 0.000 }
gfCNCPoint5[9628] = {X 388.0399, Y 11.2077, Z -7.1667, A 0.000, B 0.000, C 0.000 }
gfCNCPoint5[9629] = {X 388.3654, Y 10.2777, Z -7.1667, A 0.000, B 0.000, C 0.000 }
gfCNCPoint5[9630] = {X 388.8896, Y 9.4435, Z -7.1667, A 0.000, B 0.000, C 0.000 }
gfCNCPoint5[9631] = {X 389.5863, Y 8.7468, Z -7.1667, A 0.000, B 0.000, C 0.000 }
gfCNCPoint5[9632] = {X 390.4205, Y 8.2226, Z -7.1667, A 0.000, B 0.000, C 0.000 }
gfCNCPoint5[9633] = {X 391.3505, Y 7.8971, Z -7.1667, A 0.000, B 0.000, C 0.000 }
gfCNCPoint5[9634] = {X 392.3296, Y 7.7868, Z -7.1667, A 0.000, B 0.000, C 0.000 }
gfCNCPoint5[9635] = {X 399.1118, Y 7.7868, Z -7.1667, A 0.000, B 0.000, C 0.000 }
gfCNCPoint5[9636] = {X 400.0909, Y 7.8971, Z -7.1667, A 0.000, B 0.000, C 0.000 }
gfCNCPoint5[9637] = {X 401.0208, Y 8.2226, Z -7.1667, A 0.000, B 0.000, C 0.000 }
gfCNCPoint5[9638] = {X 401.8551, Y 8.7468, Z -7.1667, A 0.000, B 0.000, C 0.000 }
gfCNCPoint5[9639] = {X 402.5518, Y 9.4435, Z -7.1667, A 0.000, B 0.000, C 0.000 }
gfCNCPoint5[9640] = {X 403.0760, Y 10.2777, Z -7.1667, A 0.000, B 0.000, C 0.000 }
gfCNCPoint5[9641] = {X 403.4014, Y 11.2077, Z -7.1667, A 0.000, B 0.000, C 0.000 }
gfCNCPoint5[9642] = {X 403.5118, Y 12.1868, Z -7.1667, A 0.000, B 0.000, C 0.000 }
gfCNCPoint5[9643] = {X 403.5115, Y 13.0233, Z -7.1667, A 0.000, B 0.000, C 0.000 }
gfCNCPoint5[9644] = {X 403.4070, Y 13.9326, Z -7.1667, A 0.000, B 0.000, C 0.000 }
gfCNCPoint5[9645] = {X 403.1165, Y 14.8007, Z -7.1667, A 0.000, B 0.000, C 0.000 }
gfCNCPoint5[9646] = {X 405.3499, Y 18.6787, Z -7.1667, A 0.000, B 0.000, C 0.000 }
gfCNCPoint5[9647] = {X 407.7805, Y 14.7418, Z -7.1667, A 0.000, B 0.000, C 0.000 }
gfCNCPoint5[9648] = {X 407.5048, Y 13.8790, Z -7.1667, A 0.000, B 0.000, C 0.000 }
gfCNCPoint5[9649] = {X 407.4115, Y 12.9780, Z -7.1667, A 0.000, B 0.000, C 0.000 }
gfCNCPoint5[9650] = {X 407.4115, Y 12.1868, Z -7.1667, A 0.000, B 0.000, C 0.000 }
gfCNCPoint5[9651] = {X 407.5219, Y 11.2077, Z -7.1667, A 0.000, B 0.000, C 0.000 }
gfCNCPoint5[9652] = {X 407.8473, Y 10.2777, Z -7.1667, A 0.000, B 0.000, C 0.000 }
gfCNCPoint5[9653] = {X 408.3715, Y 9.4435, Z -7.1667, A 0.000, B 0.000, C 0.000 }
gfCNCPoint5[9654] = {X 409.0682, Y 8.7468, Z -7.1667, A 0.000, B 0.000, C 0.000 }
gfCNCPoint5[9655] = {X 409.9024, Y 8.2226, Z -7.1667, A 0.000, B 0.000, C 0.000 }
gfCNCPoint5[9656] = {X 410.8324, Y 7.8971, Z -7.1667, A 0.000, B 0.000, C 0.000 }
gfCNCPoint5[9657] = {X 411.8115, Y 7.7868, Z -7.1667, A 0.000, B 0.000, C 0.000 }
gfCNCPoint5[9658] = {X 419.3245, Y 7.7868, Z -7.1667, A 0.000, B 0.000, C 0.000 }
gfCNCPoint5[9659] = {X 420.3036, Y 7.8971, Z -7.1667, A 0.000, B 0.000, C 0.000 }
gfCNCPoint5[9660] = {X 421.2335, Y 8.2226, Z -7.1667, A 0.000, B 0.000, C 0.000 }
gfCNCPoint5[9661] = {X 422.0678, Y 8.7468, Z -7.1667, A 0.000, B 0.000, C 0.000 }
gfCNCPoint5[9662] = {X 422.7645, Y 9.4435, Z -7.1667, A 0.000, B 0.000, C 0.000 }
gfCNCPoint5[9663] = {X 423.2887, Y 10.2777, Z -7.1667, A 0.000, B 0.000, C 0.000 }
gfCNCPoint5[9664] = {X 423.6141, Y 11.2077, Z -7.1667, A 0.000, B 0.000, C 0.000 }
gfCNCPoint5[9665] = {X 423.7245, Y 12.1868, Z -7.1667, A 0.000, B 0.000, C 0.000 }
gfCNCPoint5[9666] = {X 423.7245, Y 12.9806, Z -7.1667, A 0.000, B 0.000, C 0.000 }
gfCNCPoint5[9667] = {X 423.6311, Y 13.8595, Z -7.1667, A 0.000, B 0.000, C 0.000 }
gfCNCPoint5[9668] = {X 423.3662, Y 14.7028, Z -7.1667, A 0.000, B 0.000, C 0.000 }
gfCNCPoint5[9669] = {X 422.9403, Y 15.4772, Z -7.1667, A 0.000, B 0.000, C 0.000 }
